(* Logix 5000 project; controller Receptivo vendor 1 type 14 code 106 rev 30.11; software revision 30.00; part 2 of 10 *)

        [54].Fecha.Minuto := 54, [54].Fecha.Segundo := 41, [54].Fecha.Milisegundos := 45401, [54].Lote := 147, [54].Operador := 5, [54].Descripcion := 'Alegria Caja 6 x 3000 cm3  - Costa', [54].EAN14 := '17702161043987', [54].QAD := '600300', [54].Peso_Real := 516.0, [54].Peso_Teorico := 519.0, [54].No_Cajas := 30, [54].Consec := 188, [54].Envase := 3000, [54].Envases_x_Caja := 6, [54].Densidad_Medida := 0.9152, [54].Linea := 3, [55].Fecha.year := 2021, [55].Fecha.Mes := 5, [55].Fecha.Dia := 27, [55].Fecha.Hora := 19, [55].Fecha.Minuto := 57, [55].Fecha.Segundo := 29, [55].Fecha.Milisegundos := 629132, [55].Lote := 147, [55].Operador := 5, [55].Descripcion := 'Alegria Caja 6 x 3000 cm3  - Costa', [55].EAN14 := '17702161043987', [55].QAD := '600300', [55].Peso_Real := 516.0, [55].Peso_Teorico := 519.0, [55].No_Cajas := 30, [55].Consec := 189, [55].Envase := 3000, [55].Envases_x_Caja := 6, [55].Densidad_Medida := 0.9152, [55].Linea := 3, [56].Fecha.year := 2021, [56].Fecha.Mes := 5, [56].Fecha.Dia := 27, [56].Fecha.Hora := 20, [56].Fecha.Segundo := 42, [56].Fecha.Milisegundos := 662176, [56].Lote := 147, [56].Operador := 5, [56].Descripcion := 'Alegria Caja 6 x 3000 cm3  - Costa', [56].EAN14 := '17702161043987', [56].QAD := '600300', [56].Peso_Real := 518.0, [56].Peso_Teorico := 519.0, [56].No_Cajas := 30, [56].Consec := 190, [56].Envase := 3000, [56].Envases_x_Caja := 6, [56].Densidad_Medida := 0.9152, [56].Linea := 3, [57].Fecha.year := 2021, [57].Fecha.Mes := 5, [57].Fecha.Dia := 27, [57].Fecha.Hora := 20, [57].Fecha.Minuto := 5,
        [57].Fecha.Segundo := 2, [57].Fecha.Milisegundos := 990759, [57].Lote := 147, [57].Operador := 5, [57].Descripcion := 'Alegria Caja 6 x 3000 cm3  - Costa', [57].EAN14 := '17702161043987', [57].QAD := '600300', [57].Peso_Real := 518.0, [57].Peso_Teorico := 519.0, [57].No_Cajas := 30, [57].Consec := 191, [57].Envase := 3000, [57].Envases_x_Caja := 6, [57].Densidad_Medida := 0.9152, [57].Linea := 3, [58].Fecha.year := 2021, [58].Fecha.Mes := 5, [58].Fecha.Dia := 27, [58].Fecha.Hora := 20, [58].Fecha.Minuto := 7, [58].Fecha.Segundo := 7, [58].Fecha.Milisegundos := 884753, [58].Lote := 147, [58].Operador := 5, [58].Descripcion := 'Alegria Caja 6 x 3000 cm3  - Costa', [58].EAN14 := '17702161043987', [58].QAD := '600300', [58].Peso_Real := 52.0, [58].Peso_Teorico := 52.0, [58].No_Cajas := 3, [58].Consec := 192, [58].Envase := 3000, [58].Envases_x_Caja := 6, [58].Densidad_Medida := 0.9152, [58].Linea := 3);
   Cola_Estacion_4 : UDT_COLA[100] := ([0].Fecha.year := 2021, [0].Fecha.Mes := 5, [0].Fecha.Dia := 28, [0].Fecha.Hora := 8, [0].Fecha.Minuto := 20, [0].Fecha.Segundo := 37, [0].Fecha.Milisegundos := 69124, [0].Lote := 148, [0].Operador := 6, [0].Descripcion := 'Aceite Vegetal Torino  Exp.', [0].EAN14 := '17702161820113', [0].QAD := '607020', [0].Peso_Real := 790.0, [0].Peso_Teorico := 786.0, [0].No_Cajas := 48, [0].Consec := 1, [0].Envase := 17250, [0].Envases_x_Caja := 1, [0].Densidad_Medida := 0.9148, [0].Linea := 5, [1].Fecha.year := 2021, [1].Fecha.Mes := 5, [1].Fecha.Dia := 28, [1].Fecha.Hora := 8, [1].Fecha.Minuto := 26, [1].Fecha.Segundo := 16, [1].Fecha.Milisegundos := 465551, [1].Lote := 148, [1].Operador := 6, [1].Descripcion := 'Aceite Vegetal Torino  Exp.', [1].EAN14 := '17702161820113', [1].QAD := '607020', [1].Peso_Real := 787.0, [1].Peso_Teorico := 786.0, [1].No_Cajas := 48, [1].Consec := 2, [1].Envase := 17250, [1].Envases_x_Caja := 1, [1].Densidad_Medida := 0.9148, [1].Linea := 5, [2].Fecha.year := 2021, [2].Fecha.Mes := 5, [2].Fecha.Dia := 28, [2].Fecha.Hora := 8, [2].Fecha.Minuto := 31, [2].Fecha.Segundo := 21, [2].Fecha.Milisegundos := 483752, [2].Lote := 148, [2].Operador := 6, [2].Descripcion := 'Aceite Vegetal Torino  Exp.', [2].EAN14 := '17702161820113', [2].QAD := '607020', [2].Peso_Real := 789.0, [2].Peso_Teorico := 786.0, [2].No_Cajas := 48, [2].Consec := 3, [2].Envase := 17250, [2].Envases_x_Caja := 1, [2].Densidad_Medida := 0.9148, [2].Linea := 5,
        [3].Fecha.year := 2021, [3].Fecha.Mes := 5, [3].Fecha.Dia := 28, [3].Fecha.Hora := 8, [3].Fecha.Minuto := 36, [3].Fecha.Segundo := 10, [3].Fecha.Milisegundos := 577902, [3].Lote := 148, [3].Operador := 6, [3].Descripcion := 'Aceite Vegetal Torino  Exp.', [3].EAN14 := '17702161820113', [3].QAD := '607020', [3].Peso_Real := 786.0, [3].Peso_Teorico := 786.0, [3].No_Cajas := 48, [3].Consec := 4, [3].Envase := 17250, [3].Envases_x_Caja := 1, [3].Densidad_Medida := 0.9148, [3].Linea := 5, [4].Fecha.year := 2021, [4].Fecha.Mes := 5, [4].Fecha.Dia := 28, [4].Fecha.Hora := 8, [4].Fecha.Minuto := 40, [4].Fecha.Segundo := 51, [4].Fecha.Milisegundos := 336954, [4].Lote := 148, [4].Operador := 6, [4].Descripcion := 'Aceite Vegetal Torino  Exp.', [4].EAN14 := '17702161820113', [4].QAD := '607020', [4].Peso_Real := 790.0, [4].Peso_Teorico := 786.0, [4].No_Cajas := 48, [4].Consec := 5, [4].Envase := 17250, [4].Envases_x_Caja := 1, [4].Densidad_Medida := 0.9148, [4].Linea := 5, [5].Fecha.year := 2021, [5].Fecha.Mes := 5, [5].Fecha.Dia := 28, [5].Fecha.Hora := 8, [5].Fecha.Minuto := 47, [5].Fecha.Segundo := 15, [5].Fecha.Milisegundos := 315402, [5].Lote := 148, [5].Operador := 6, [5].Descripcion := 'Aceite Vegetal Torino  Exp.', [5].EAN14 := '17702161820113', [5].QAD := '607020', [5].Peso_Real := 789.0, [5].Peso_Teorico := 786.0, [5].No_Cajas := 48, [5].Consec := 6, [5].Envase := 17250, [5].Envases_x_Caja := 1, [5].Densidad_Medida := 0.9148, [5].Linea := 5,
        [6].Fecha.year := 2021, [6].Fecha.Mes := 5, [6].Fecha.Dia := 28, [6].Fecha.Hora := 8, [6].Fecha.Minuto := 52, [6].Fecha.Segundo := 9, [6].Fecha.Milisegundos := 719173, [6].Lote := 148, [6].Operador := 6, [6].Descripcion := 'Aceite Vegetal Torino  Exp.', [6].EAN14 := '17702161820113', [6].QAD := '607020', [6].Peso_Real := 787.0, [6].Peso_Teorico := 786.0, [6].No_Cajas := 48, [6].Consec := 7, [6].Envase := 17250, [6].Envases_x_Caja := 1, [6].Densidad_Medida := 0.9148, [6].Linea := 5, [7].Fecha.year := 2021, [7].Fecha.Mes := 5, [7].Fecha.Dia := 28, [7].Fecha.Hora := 8, [7].Fecha.Minuto := 55, [7].Fecha.Segundo := 40, [7].Fecha.Milisegundos := 508565, [7].Lote := 148, [7].Operador := 6, [7].Descripcion := 'Aceite Vegetal Torino  Exp.', [7].EAN14 := '17702161820113', [7].QAD := '607020', [7].Peso_Real := 791.0, [7].Peso_Teorico := 786.0, [7].No_Cajas := 48, [7].Consec := 8, [7].Envase := 17250, [7].Envases_x_Caja := 1, [7].Densidad_Medida := 0.9148, [7].Linea := 5, [8].Fecha.year := 2021, [8].Fecha.Mes := 5, [8].Fecha.Dia := 28, [8].Fecha.Hora := 9, [8].Fecha.Segundo := 2, [8].Fecha.Milisegundos := 670788, [8].Lote := 148, [8].Operador := 6, [8].Descripcion := 'Aceite Vegetal Torino  Exp.', [8].EAN14 := '17702161820113', [8].QAD := '607020', [8].Peso_Real := 789.0, [8].Peso_Teorico := 786.0, [8].No_Cajas := 48, [8].Consec := 9, [8].Envase := 17250, [8].Envases_x_Caja := 1, [8].Densidad_Medida := 0.9148, [8].Linea := 5, [9].Fecha.year := 2021,
        [9].Fecha.Mes := 5, [9].Fecha.Dia := 28, [9].Fecha.Hora := 9, [9].Fecha.Minuto := 4, [9].Fecha.Segundo := 22, [9].Fecha.Milisegundos := 670540, [9].Lote := 148, [9].Operador := 6, [9].Descripcion := 'Aceite Vegetal Torino  Exp.', [9].EAN14 := '17702161820113', [9].QAD := '607020', [9].Peso_Real := 788.0, [9].Peso_Teorico := 786.0, [9].No_Cajas := 48, [9].Consec := 10, [9].Envase := 17250, [9].Envases_x_Caja := 1, [9].Densidad_Medida := 0.9148, [9].Linea := 5, [10].Fecha.year := 2021, [10].Fecha.Mes := 5, [10].Fecha.Dia := 28, [10].Fecha.Hora := 9, [10].Fecha.Minuto := 12, [10].Fecha.Segundo := 17, [10].Fecha.Milisegundos := 553199, [10].Lote := 148, [10].Operador := 6, [10].Descripcion := 'Aceite Vegetal Torino  Exp.', [10].EAN14 := '17702161820113', [10].QAD := '607020', [10].Peso_Real := 787.0, [10].Peso_Teorico := 786.0, [10].No_Cajas := 48, [10].Consec := 11, [10].Envase := 17250, [10].Envases_x_Caja := 1, [10].Densidad_Medida := 0.9148, [10].Linea := 5, [11].Fecha.year := 2021, [11].Fecha.Mes := 5, [11].Fecha.Dia := 28, [11].Fecha.Hora := 9, [11].Fecha.Minuto := 17, [11].Fecha.Segundo := 9, [11].Fecha.Milisegundos := 930477, [11].Lote := 148, [11].Operador := 6, [11].Descripcion := 'Aceite Vegetal Torino  Exp.', [11].EAN14 := '17702161820113', [11].QAD := '607020', [11].Peso_Real := 787.0, [11].Peso_Teorico := 786.0, [11].No_Cajas := 48, [11].Consec := 12, [11].Envase := 17250, [11].Envases_x_Caja := 1, [11].Densidad_Medida := 0.9148, [11].Linea := 5, [12].Fecha.year := 2021,
        [12].Fecha.Mes := 5, [12].Fecha.Dia := 28, [12].Fecha.Hora := 9, [12].Fecha.Minuto := 21, [12].Fecha.Segundo := 57, [12].Fecha.Milisegundos := 591967, [12].Lote := 148, [12].Operador := 6, [12].Descripcion := 'Aceite Vegetal Torino  Exp.', [12].EAN14 := '17702161820113', [12].QAD := '607020', [12].Peso_Real := 787.0, [12].Peso_Teorico := 786.0, [12].No_Cajas := 48, [12].Consec := 13, [12].Envase := 17250, [12].Envases_x_Caja := 1, [12].Densidad_Medida := 0.9148, [12].Linea := 5, [13].Fecha.year := 2021, [13].Fecha.Mes := 5, [13].Fecha.Dia := 28, [13].Fecha.Hora := 9, [13].Fecha.Minuto := 26, [13].Fecha.Segundo := 49, [13].Fecha.Milisegundos := 73835, [13].Lote := 148, [13].Operador := 6, [13].Descripcion := 'Aceite Vegetal Torino  Exp.', [13].EAN14 := '17702161820113', [13].QAD := '607020', [13].Peso_Real := 786.0, [13].Peso_Teorico := 786.0, [13].No_Cajas := 48, [13].Consec := 14, [13].Envase := 17250, [13].Envases_x_Caja := 1, [13].Densidad_Medida := 0.9148, [13].Linea := 5, [14].Fecha.year := 2021, [14].Fecha.Mes := 5, [14].Fecha.Dia := 28, [14].Fecha.Hora := 9, [14].Fecha.Minuto := 32, [14].Fecha.Segundo := 14, [14].Fecha.Milisegundos := 130378, [14].Lote := 148, [14].Operador := 6, [14].Descripcion := 'Aceite Vegetal Torino  Exp.', [14].EAN14 := '17702161820113', [14].QAD := '607020', [14].Peso_Real := 786.0, [14].Peso_Teorico := 786.0, [14].No_Cajas := 48, [14].Consec := 15, [14].Envase := 17250, [14].Envases_x_Caja := 1, [14].Densidad_Medida := 0.9148, [14].Linea := 5, [15].Fecha.year := 2021,
        [15].Fecha.Mes := 5, [15].Fecha.Dia := 28, [15].Fecha.Hora := 9, [15].Fecha.Minuto := 38, [15].Fecha.Segundo := 57, [15].Fecha.Milisegundos := 869726, [15].Lote := 148, [15].Operador := 6, [15].Descripcion := 'Aceite Vegetal Torino  Exp.', [15].EAN14 := '17702161820113', [15].QAD := '607020', [15].Peso_Real := 789.0, [15].Peso_Teorico := 786.0, [15].No_Cajas := 48, [15].Consec := 16, [15].Envase := 17250, [15].Envases_x_Caja := 1, [15].Densidad_Medida := 0.9148, [15].Linea := 5, [16].Fecha.year := 2021, [16].Fecha.Mes := 5, [16].Fecha.Dia := 28, [16].Fecha.Hora := 9, [16].Fecha.Minuto := 43, [16].Fecha.Segundo := 25, [16].Fecha.Milisegundos := 20130, [16].Lote := 148, [16].Operador := 6, [16].Descripcion := 'Aceite Vegetal Torino  Exp.', [16].EAN14 := '17702161820113', [16].QAD := '607020', [16].Peso_Real := 790.0, [16].Peso_Teorico := 786.0, [16].No_Cajas := 48, [16].Consec := 17, [16].Envase := 17250, [16].Envases_x_Caja := 1, [16].Densidad_Medida := 0.9148, [16].Linea := 5, [17].Fecha.year := 2021, [17].Fecha.Mes := 5, [17].Fecha.Dia := 28, [17].Fecha.Hora := 9, [17].Fecha.Minuto := 47, [17].Fecha.Segundo := 58, [17].Fecha.Milisegundos := 358560, [17].Lote := 148, [17].Operador := 6, [17].Descripcion := 'Aceite Vegetal Torino  Exp.', [17].EAN14 := '17702161820113', [17].QAD := '607020', [17].Peso_Real := 789.0, [17].Peso_Teorico := 786.0, [17].No_Cajas := 48, [17].Consec := 18, [17].Envase := 17250, [17].Envases_x_Caja := 1, [17].Densidad_Medida := 0.9148, [17].Linea := 5, [18].Fecha.year := 2021,
        [18].Fecha.Mes := 5, [18].Fecha.Dia := 28, [18].Fecha.Hora := 9, [18].Fecha.Minuto := 51, [18].Fecha.Segundo := 17, [18].Fecha.Milisegundos := 179162, [18].Lote := 148, [18].Operador := 6, [18].Descripcion := 'Aceite Vegetal Torino  Exp.', [18].EAN14 := '17702161820113', [18].QAD := '607020', [18].Peso_Real := 788.0, [18].Peso_Teorico := 786.0, [18].No_Cajas := 48, [18].Consec := 19, [18].Envase := 17250, [18].Envases_x_Caja := 1, [18].Densidad_Medida := 0.9148, [18].Linea := 5, [19].Fecha.year := 2021, [19].Fecha.Mes := 5, [19].Fecha.Dia := 28, [19].Fecha.Hora := 9, [19].Fecha.Minuto := 54, [19].Fecha.Segundo := 47, [19].Fecha.Milisegundos := 964537, [19].Lote := 148, [19].Operador := 6, [19].Descripcion := 'Aceite Vegetal Torino  Exp.', [19].EAN14 := '17702161820113', [19].QAD := '607020', [19].Peso_Real := 788.0, [19].Peso_Teorico := 786.0, [19].No_Cajas := 48, [19].Consec := 20, [19].Envase := 17250, [19].Envases_x_Caja := 1, [19].Densidad_Medida := 0.9148, [19].Linea := 5, [20].Fecha.year := 2021, [20].Fecha.Mes := 5, [20].Fecha.Dia := 28, [20].Fecha.Hora := 10, [20].Fecha.Minuto := 3, [20].Fecha.Segundo := 29, [20].Fecha.Milisegundos := 988763, [20].Lote := 148, [20].Operador := 6, [20].Descripcion := 'Aceite Vegetal Torino  Exp.', [20].EAN14 := '17702161820113', [20].QAD := '607020', [20].Peso_Real := 787.0, [20].Peso_Teorico := 786.0, [20].No_Cajas := 48, [20].Consec := 21, [20].Envase := 17250, [20].Envases_x_Caja := 1, [20].Densidad_Medida := 0.9148, [20].Linea := 5, [21].Fecha.year := 2021,
        [21].Fecha.Mes := 5, [21].Fecha.Dia := 28, [21].Fecha.Hora := 10, [21].Fecha.Minuto := 9, [21].Fecha.Segundo := 7, [21].Fecha.Milisegundos := 475825, [21].Lote := 148, [21].Operador := 6, [21].Descripcion := 'Aceite Vegetal Torino  Exp.', [21].EAN14 := '17702161820113', [21].QAD := '607020', [21].Peso_Real := 788.0, [21].Peso_Teorico := 786.0, [21].No_Cajas := 48, [21].Consec := 22, [21].Envase := 17250, [21].Envases_x_Caja := 1, [21].Densidad_Medida := 0.9148, [21].Linea := 5, [22].Fecha.year := 2021, [22].Fecha.Mes := 5, [22].Fecha.Dia := 28, [22].Fecha.Hora := 10, [22].Fecha.Minuto := 13, [22].Fecha.Segundo := 59, [22].Fecha.Milisegundos := 393945, [22].Lote := 148, [22].Operador := 6, [22].Descripcion := 'Aceite Vegetal Torino  Exp.', [22].EAN14 := '17702161820113', [22].QAD := '607020', [22].Peso_Real := 788.0, [22].Peso_Teorico := 786.0, [22].No_Cajas := 48, [22].Consec := 23, [22].Envase := 17250, [22].Envases_x_Caja := 1, [22].Densidad_Medida := 0.9148, [22].Linea := 5, [23].Fecha.year := 2021, [23].Fecha.Mes := 5, [23].Fecha.Dia := 28, [23].Fecha.Hora := 10, [23].Fecha.Minuto := 18, [23].Fecha.Segundo := 56, [23].Fecha.Milisegundos := 553433, [23].Lote := 148, [23].Operador := 6, [23].Descripcion := 'Aceite Vegetal Torino  Exp.', [23].EAN14 := '17702161820113', [23].QAD := '607020', [23].Peso_Real := 787.0, [23].Peso_Teorico := 786.0, [23].No_Cajas := 48, [23].Consec := 24, [23].Envase := 17250, [23].Envases_x_Caja := 1, [23].Densidad_Medida := 0.9148, [23].Linea := 5, [24].Fecha.year := 2021,
        [24].Fecha.Mes := 5, [24].Fecha.Dia := 28, [24].Fecha.Hora := 10, [24].Fecha.Minuto := 24, [24].Fecha.Segundo := 26, [24].Fecha.Milisegundos := 21235, [24].Lote := 148, [24].Operador := 6, [24].Descripcion := 'Aceite Vegetal Torino  Exp.', [24].EAN14 := '17702161820113', [24].QAD := '607020', [24].Peso_Real := 787.0, [24].Peso_Teorico := 786.0, [24].No_Cajas := 48, [24].Consec := 25, [24].Envase := 17250, [24].Envases_x_Caja := 1, [24].Densidad_Medida := 0.9148, [24].Linea := 5, [25].Fecha.year := 2021, [25].Fecha.Mes := 5, [25].Fecha.Dia := 28, [25].Fecha.Hora := 10, [25].Fecha.Minuto := 30, [25].Fecha.Segundo := 54, [25].Fecha.Milisegundos := 336113, [25].Lote := 148, [25].Operador := 6, [25].Descripcion := 'Aceite Vegetal Torino  Exp.', [25].EAN14 := '17702161820113', [25].QAD := '607020', [25].Peso_Real := 790.0, [25].Peso_Teorico := 786.0, [25].No_Cajas := 48, [25].Consec := 26, [25].Envase := 17250, [25].Envases_x_Caja := 1, [25].Densidad_Medida := 0.9148, [25].Linea := 5, [26].Fecha.year := 2021, [26].Fecha.Mes := 5, [26].Fecha.Dia := 28, [26].Fecha.Hora := 10, [26].Fecha.Minuto := 35, [26].Fecha.Segundo := 32, [26].Fecha.Milisegundos := 418041, [26].Lote := 148, [26].Operador := 6, [26].Descripcion := 'Aceite Vegetal Torino  Exp.', [26].EAN14 := '17702161820113', [26].QAD := '607020', [26].Peso_Real := 789.0, [26].Peso_Teorico := 786.0, [26].No_Cajas := 48, [26].Consec := 27, [26].Envase := 17250, [26].Envases_x_Caja := 1, [26].Densidad_Medida := 0.9148, [26].Linea := 5, [27].Fecha.year := 2021,
        [27].Fecha.Mes := 5, [27].Fecha.Dia := 28, [27].Fecha.Hora := 10, [27].Fecha.Minuto := 40, [27].Fecha.Segundo := 38, [27].Fecha.Milisegundos := 622882, [27].Lote := 148, [27].Operador := 6, [27].Descripcion := 'Aceite Vegetal Torino  Exp.', [27].EAN14 := '17702161820113', [27].QAD := '607020', [27].Peso_Real := 794.0, [27].Peso_Teorico := 786.0, [27].No_Cajas := 48, [27].Consec := 28, [27].Envase := 17250, [27].Envases_x_Caja := 1, [27].Densidad_Medida := 0.9148, [27].Linea := 5, [28].Fecha.year := 2021, [28].Fecha.Mes := 5, [28].Fecha.Dia := 28, [28].Fecha.Hora := 10, [28].Fecha.Minuto := 45, [28].Fecha.Segundo := 3, [28].Fecha.Milisegundos := 533526, [28].Lote := 148, [28].Operador := 6, [28].Descripcion := 'Aceite Vegetal Torino  Exp.', [28].EAN14 := '17702161820113', [28].QAD := '607020', [28].Peso_Real := 791.0, [28].Peso_Teorico := 786.0, [28].No_Cajas := 48, [28].Consec := 29, [28].Envase := 17250, [28].Envases_x_Caja := 1, [28].Densidad_Medida := 0.9148, [28].Linea := 5, [29].Fecha.year := 2021, [29].Fecha.Mes := 5, [29].Fecha.Dia := 28, [29].Fecha.Hora := 10, [29].Fecha.Minuto := 49, [29].Fecha.Segundo := 29, [29].Fecha.Milisegundos := 771525, [29].Lote := 148, [29].Operador := 6, [29].Descripcion := 'Aceite Vegetal Torino  Exp.', [29].EAN14 := '17702161820113', [29].QAD := '607020', [29].Peso_Real := 789.0, [29].Peso_Teorico := 786.0, [29].No_Cajas := 48, [29].Consec := 30, [29].Envase := 17250, [29].Envases_x_Caja := 1, [29].Densidad_Medida := 0.9148, [29].Linea := 5, [30].Fecha.year := 2021,
        [30].Fecha.Mes := 5, [30].Fecha.Dia := 28, [30].Fecha.Hora := 11, [30].Fecha.Minuto := 38, [30].Fecha.Segundo := 27, [30].Fecha.Milisegundos := 412017, [30].Lote := 148, [30].Operador := 6, [30].Descripcion := 'Aceite Vegetal Torino  Exp.', [30].EAN14 := '17702161820113', [30].QAD := '607020', [30].Peso_Real := 787.0, [30].Peso_Teorico := 786.0, [30].No_Cajas := 48, [30].Consec := 37, [30].Envase := 17250, [30].Envases_x_Caja := 1, [30].Densidad_Medida := 0.9148, [30].Linea := 5, [31].Fecha.year := 2021, [31].Fecha.Mes := 5, [31].Fecha.Dia := 28, [31].Fecha.Hora := 11, [31].Fecha.Minuto := 43, [31].Fecha.Segundo := 1, [31].Fecha.Milisegundos := 735545, [31].Lote := 148, [31].Operador := 6, [31].Descripcion := 'Aceite Vegetal Torino  Exp.', [31].EAN14 := '17702161820113', [31].QAD := '607020', [31].Peso_Real := 787.0, [31].Peso_Teorico := 786.0, [31].No_Cajas := 48, [31].Consec := 39, [31].Envase := 17250, [31].Envases_x_Caja := 1, [31].Densidad_Medida := 0.9148, [31].Linea := 5, [32].Fecha.year := 2021, [32].Fecha.Mes := 5, [32].Fecha.Dia := 28, [32].Fecha.Hora := 11, [32].Fecha.Minuto := 47, [32].Fecha.Segundo := 48, [32].Fecha.Milisegundos := 728105, [32].Lote := 148, [32].Operador := 6, [32].Descripcion := 'Aceite Vegetal Torino  Exp.', [32].EAN14 := '17702161820113', [32].QAD := '607020', [32].Peso_Real := 787.0, [32].Peso_Teorico := 786.0, [32].No_Cajas := 48, [32].Consec := 42, [32].Envase := 17250, [32].Envases_x_Caja := 1, [32].Densidad_Medida := 0.9148, [32].Linea := 5, [33].Fecha.year := 2021,
        [33].Fecha.Mes := 5, [33].Fecha.Dia := 28, [33].Fecha.Hora := 11, [33].Fecha.Minuto := 54, [33].Fecha.Segundo := 28, [33].Fecha.Milisegundos := 332631, [33].Lote := 148, [33].Operador := 6, [33].Descripcion := 'Aceite Vegetal Torino  Exp.', [33].EAN14 := '17702161820113', [33].QAD := '607020', [33].Peso_Real := 788.0, [33].Peso_Teorico := 786.0, [33].No_Cajas := 48, [33].Consec := 46, [33].Envase := 17250, [33].Envases_x_Caja := 1, [33].Densidad_Medida := 0.9148, [33].Linea := 5, [34].Fecha.year := 2021, [34].Fecha.Mes := 5, [34].Fecha.Dia := 28, [34].Fecha.Hora := 12, [34].Fecha.Minuto := 37, [34].Fecha.Segundo := 29, [34].Fecha.Milisegundos := 409886, [34].Lote := 148, [34].Operador := 6, [34].Descripcion := 'Aceite Vegetal Torino  Exp.', [34].EAN14 := '17702161820113', [34].QAD := '607020', [34].Peso_Real := 789.0, [34].Peso_Teorico := 786.0, [34].No_Cajas := 48, [34].Consec := 61, [34].Envase := 17250, [34].Envases_x_Caja := 1, [34].Densidad_Medida := 0.9148, [34].Linea := 5, [35].Fecha.year := 2021, [35].Fecha.Mes := 5, [35].Fecha.Dia := 28, [35].Fecha.Hora := 12, [35].Fecha.Minuto := 48, [35].Fecha.Segundo := 16, [35].Fecha.Milisegundos := 558137, [35].Lote := 148, [35].Operador := 6, [35].Descripcion := 'Aceite Vegetal Torino  Exp.', [35].EAN14 := '17702161820113', [35].QAD := '607020', [35].Peso_Real := 788.0, [35].Peso_Teorico := 786.0, [35].No_Cajas := 48, [35].Consec := 64, [35].Envase := 17250, [35].Envases_x_Caja := 1, [35].Densidad_Medida := 0.9148, [35].Linea := 5, [36].Fecha.year := 2021,
        [36].Fecha.Mes := 5, [36].Fecha.Dia := 28, [36].Fecha.Hora := 12, [36].Fecha.Minuto := 53, [36].Fecha.Segundo := 29, [36].Fecha.Milisegundos := 332540, [36].Lote := 148, [36].Operador := 6, [36].Descripcion := 'Aceite Vegetal Torino  Exp.', [36].EAN14 := '17702161820113', [36].QAD := '607020', [36].Peso_Real := 790.0, [36].Peso_Teorico := 786.0, [36].No_Cajas := 48, [36].Consec := 66, [36].Envase := 17250, [36].Envases_x_Caja := 1, [36].Densidad_Medida := 0.9148, [36].Linea := 5, [37].Fecha.year := 2021, [37].Fecha.Mes := 5, [37].Fecha.Dia := 28, [37].Fecha.Hora := 12, [37].Fecha.Minuto := 59, [37].Fecha.Segundo := 39, [37].Fecha.Milisegundos := 67313, [37].Lote := 148, [37].Operador := 6, [37].Descripcion := 'Aceite Vegetal Torino  Exp.', [37].EAN14 := '17702161820113', [37].QAD := '607020', [37].Peso_Real := 784.0, [37].Peso_Teorico := 786.0, [37].No_Cajas := 48, [37].Consec := 68, [37].Envase := 17250, [37].Envases_x_Caja := 1, [37].Densidad_Medida := 0.9148, [37].Linea := 5, [38].Fecha.year := 2021, [38].Fecha.Mes := 5, [38].Fecha.Dia := 28, [38].Fecha.Hora := 13, [38].Fecha.Minuto := 4, [38].Fecha.Segundo := 44, [38].Fecha.Milisegundos := 914365, [38].Lote := 148, [38].Operador := 6, [38].Descripcion := 'Aceite Vegetal Torino  Exp.', [38].EAN14 := '17702161820113', [38].QAD := '607020', [38].Peso_Real := 788.0, [38].Peso_Teorico := 786.0, [38].No_Cajas := 48, [38].Consec := 70, [38].Envase := 17250, [38].Envases_x_Caja := 1, [38].Densidad_Medida := 0.9148, [38].Linea := 5, [39].Fecha.year := 2021,
        [39].Fecha.Mes := 5, [39].Fecha.Dia := 28, [39].Fecha.Hora := 13, [39].Fecha.Minuto := 9, [39].Fecha.Segundo := 50, [39].Fecha.Milisegundos := 10253, [39].Lote := 148, [39].Operador := 6, [39].Descripcion := 'Aceite Vegetal Torino  Exp.', [39].EAN14 := '17702161820113', [39].QAD := '607020', [39].Peso_Real := 788.0, [39].Peso_Teorico := 786.0, [39].No_Cajas := 48, [39].Consec := 73, [39].Envase := 17250, [39].Envases_x_Caja := 1, [39].Densidad_Medida := 0.9148, [39].Linea := 5, [40].Fecha.year := 2021, [40].Fecha.Mes := 5, [40].Fecha.Dia := 28, [40].Fecha.Hora := 13, [40].Fecha.Minuto := 18, [40].Fecha.Segundo := 54, [40].Fecha.Milisegundos := 825126, [40].Lote := 148, [40].Operador := 6, [40].Descripcion := 'Aceite Vegetal Torino  Exp.', [40].EAN14 := '17702161820113', [40].QAD := '607020', [40].Peso_Real := 790.0, [40].Peso_Teorico := 786.0, [40].No_Cajas := 48, [40].Consec := 78, [40].Envase := 17250, [40].Envases_x_Caja := 1, [40].Densidad_Medida := 0.9148, [40].Linea := 5, [41].Fecha.year := 2021, [41].Fecha.Mes := 5, [41].Fecha.Dia := 28, [41].Fecha.Hora := 13, [41].Fecha.Minuto := 23, [41].Fecha.Segundo := 24, [41].Fecha.Milisegundos := 204408, [41].Lote := 148, [41].Operador := 6, [41].Descripcion := 'Aceite Vegetal Torino  Exp.', [41].EAN14 := '17702161820113', [41].QAD := '607020', [41].Peso_Real := 790.0, [41].Peso_Teorico := 786.0, [41].No_Cajas := 48, [41].Consec := 81, [41].Envase := 17250, [41].Envases_x_Caja := 1, [41].Densidad_Medida := 0.9148, [41].Linea := 5, [42].Fecha.year := 2021,
        [42].Fecha.Mes := 5, [42].Fecha.Dia := 28, [42].Fecha.Hora := 13, [42].Fecha.Minuto := 28, [42].Fecha.Segundo := 7, [42].Fecha.Milisegundos := 125838, [42].Lote := 148, [42].Operador := 6, [42].Descripcion := 'Aceite Vegetal Torino  Exp.', [42].EAN14 := '17702161820113', [42].QAD := '607020', [42].Peso_Real := 787.0, [42].Peso_Teorico := 786.0, [42].No_Cajas := 48, [42].Consec := 84, [42].Envase := 17250, [42].Envases_x_Caja := 1, [42].Densidad_Medida := 0.9148, [42].Linea := 5, [43].Fecha.year := 2021, [43].Fecha.Mes := 5, [43].Fecha.Dia := 28, [43].Fecha.Hora := 13, [43].Fecha.Minuto := 34, [43].Fecha.Segundo := 9, [43].Fecha.Milisegundos := 399329, [43].Lote := 148, [43].Operador := 6, [43].Descripcion := 'Aceite Vegetal Torino  Exp.', [43].EAN14 := '17702161820113', [43].QAD := '607020', [43].Peso_Real := 788.0, [43].Peso_Teorico := 786.0, [43].No_Cajas := 48, [43].Consec := 87, [43].Envase := 17250, [43].Envases_x_Caja := 1, [43].Densidad_Medida := 0.9148, [43].Linea := 5, [44].Fecha.year := 2021, [44].Fecha.Mes := 5, [44].Fecha.Dia := 28, [44].Fecha.Hora := 13, [44].Fecha.Minuto := 42, [44].Fecha.Segundo := 2, [44].Fecha.Milisegundos := 643055, [44].Lote := 148, [44].Operador := 6, [44].Descripcion := 'Aceite Vegetal Torino  Exp.', [44].EAN14 := '17702161820113', [44].QAD := '607020', [44].Peso_Real := 791.0, [44].Peso_Teorico := 786.0, [44].No_Cajas := 48, [44].Consec := 88, [44].Envase := 17250, [44].Envases_x_Caja := 1, [44].Densidad_Medida := 0.9148, [44].Linea := 5, [45].Fecha.year := 2021,
        [45].Fecha.Mes := 5, [45].Fecha.Dia := 28, [45].Fecha.Hora := 13, [45].Fecha.Minuto := 54, [45].Fecha.Segundo := 53, [45].Fecha.Milisegundos := 530969, [45].Lote := 148, [45].Operador := 6, [45].Descripcion := 'Aceite Vegetal Torino  Exp.', [45].EAN14 := '17702161820113', [45].QAD := '607020', [45].Peso_Real := 792.0, [45].Peso_Teorico := 786.0, [45].No_Cajas := 48, [45].Consec := 90, [45].Envase := 17250, [45].Envases_x_Caja := 1, [45].Densidad_Medida := 0.9148, [45].Linea := 5, [46].Fecha.year := 2021, [46].Fecha.Mes := 5, [46].Fecha.Dia := 28, [46].Fecha.Hora := 14, [46].Fecha.Minuto := 1, [46].Fecha.Segundo := 32, [46].Fecha.Milisegundos := 314203, [46].Lote := 148, [46].Operador := 6, [46].Descripcion := 'Aceite Vegetal Torino  Exp.', [46].EAN14 := '17702161820113', [46].QAD := '607020', [46].Peso_Real := 786.0, [46].Peso_Teorico := 786.0, [46].No_Cajas := 48, [46].Consec := 94, [46].Envase := 17250, [46].Envases_x_Caja := 1, [46].Densidad_Medida := 0.9148, [46].Linea := 5, [47].Fecha.year := 2021, [47].Fecha.Mes := 5, [47].Fecha.Dia := 28, [47].Fecha.Hora := 14, [47].Fecha.Minuto := 13, [47].Fecha.Segundo := 9, [47].Fecha.Milisegundos := 540121, [47].Lote := 148, [47].Operador := 6, [47].Descripcion := 'Aceite Vegetal Torino  Exp.', [47].EAN14 := '17702161820113', [47].QAD := '607020', [47].Peso_Real := 787.0, [47].Peso_Teorico := 786.0, [47].No_Cajas := 48, [47].Consec := 98, [47].Envase := 17250, [47].Envases_x_Caja := 1, [47].Densidad_Medida := 0.9148, [47].Linea := 5, [48].Fecha.year := 2021,
        [48].Fecha.Mes := 5, [48].Fecha.Dia := 28, [48].Fecha.Hora := 14, [48].Fecha.Minuto := 20, [48].Fecha.Segundo := 32, [48].Fecha.Milisegundos := 366895, [48].Lote := 148, [48].Operador := 6, [48].Descripcion := 'Aceite Vegetal Torino  Exp.', [48].EAN14 := '17702161820113', [48].QAD := '607020', [48].Peso_Real := 788.0, [48].Peso_Teorico := 786.0, [48].No_Cajas := 48, [48].Consec := 102, [48].Envase := 17250, [48].Envases_x_Caja := 1, [48].Densidad_Medida := 0.9148, [48].Linea := 5, [49].Fecha.year := 2021, [49].Fecha.Mes := 5, [49].Fecha.Dia := 28, [49].Fecha.Hora := 14, [49].Fecha.Minuto := 25, [49].Fecha.Segundo := 56, [49].Fecha.Milisegundos := 412691, [49].Lote := 148, [49].Operador := 6, [49].Descripcion := 'Aceite Vegetal Torino  Exp.', [49].EAN14 := '17702161820113', [49].QAD := '607020', [49].Peso_Real := 789.0, [49].Peso_Teorico := 786.0, [49].No_Cajas := 48, [49].Consec := 103, [49].Envase := 17250, [49].Envases_x_Caja := 1, [49].Densidad_Medida := 0.9148, [49].Linea := 5, [50].Fecha.year := 2021, [50].Fecha.Mes := 5, [50].Fecha.Dia := 28, [50].Fecha.Hora := 14, [50].Fecha.Minuto := 34, [50].Fecha.Segundo := 53, [50].Fecha.Milisegundos := 121800, [50].Lote := 148, [50].Operador := 6, [50].Descripcion := 'Aceite Vegetal Torino  Exp.', [50].EAN14 := '17702161820113', [50].QAD := '607020', [50].Peso_Real := 786.0, [50].Peso_Teorico := 786.0, [50].No_Cajas := 48, [50].Consec := 106, [50].Envase := 17250, [50].Envases_x_Caja := 1, [50].Densidad_Medida := 0.9148, [50].Linea := 5, [51].Fecha.year := 2021,
        [51].Fecha.Mes := 5, [51].Fecha.Dia := 28, [51].Fecha.Hora := 14, [51].Fecha.Minuto := 41, [51].Fecha.Segundo := 59, [51].Fecha.Milisegundos := 904400, [51].Lote := 148, [51].Operador := 6, [51].Descripcion := 'Aceite Vegetal Torino  Exp.', [51].EAN14 := '17702161820113', [51].QAD := '607020', [51].Peso_Real := 789.0, [51].Peso_Teorico := 786.0, [51].No_Cajas := 48, [51].Consec := 108, [51].Envase := 17250, [51].Envases_x_Caja := 1, [51].Densidad_Medida := 0.9148, [51].Linea := 5, [52].Fecha.year := 2021, [52].Fecha.Mes := 5, [52].Fecha.Dia := 28, [52].Fecha.Hora := 14, [52].Fecha.Minuto := 49, [52].Fecha.Segundo := 25, [52].Fecha.Milisegundos := 216916, [52].Lote := 148, [52].Operador := 6, [52].Descripcion := 'Aceite Vegetal Torino  Exp.', [52].EAN14 := '17702161820113', [52].QAD := '607020', [52].Peso_Real := 787.0, [52].Peso_Teorico := 786.0, [52].No_Cajas := 48, [52].Consec := 110, [52].Envase := 17250, [52].Envases_x_Caja := 1, [52].Densidad_Medida := 0.9148, [52].Linea := 5);
   Cola_Estacion_4_A : UDT_COLA[100] := ([0].Fecha.year := 2021, [0].Fecha.Mes := 5, [0].Fecha.Dia := 27, [0].Fecha.Hora := 8, [0].Fecha.Minuto := 12, [0].Fecha.Segundo := 20, [0].Fecha.Milisegundos := 439054, [0].Lote := 147, [0].Operador := 6, [0].Descripcion := 'Aceite Vegetal Torino  Exp.', [0].EAN14 := '17702161820113', [0].QAD := '607020', [0].Peso_Real := 792.0, [0].Peso_Teorico := 786.0, [0].No_Cajas := 48, [0].Consec := 1, [0].Envase := 17250, [0].Envases_x_Caja := 1, [0].Densidad_Medida := 0.9148, [0].Linea := 5, [1].Fecha.year := 2021, [1].Fecha.Mes := 5, [1].Fecha.Dia := 27, [1].Fecha.Hora := 8, [1].Fecha.Minuto := 16, [1].Fecha.Segundo := 14, [1].Fecha.Milisegundos := 936761, [1].Lote := 147, [1].Operador := 6, [1].Descripcion := 'Aceite Vegetal Torino  Exp.', [1].EAN14 := '17702161820113', [1].QAD := '607020', [1].Peso_Real := 791.0, [1].Peso_Teorico := 786.0, [1].No_Cajas := 48, [1].Consec := 2, [1].Envase := 17250, [1].Envases_x_Caja := 1, [1].Densidad_Medida := 0.9148, [1].Linea := 5, [2].Fecha.year := 2021, [2].Fecha.Mes := 5, [2].Fecha.Dia := 27, [2].Fecha.Hora := 8, [2].Fecha.Minuto := 21, [2].Fecha.Segundo := 6, [2].Fecha.Milisegundos := 817817, [2].Lote := 147, [2].Operador := 6, [2].Descripcion := 'Aceite Vegetal Torino  Exp.', [2].EAN14 := '17702161820113', [2].QAD := '607020', [2].Peso_Real := 794.0, [2].Peso_Teorico := 786.0, [2].No_Cajas := 48, [2].Consec := 3, [2].Envase := 17250, [2].Envases_x_Caja := 1, [2].Densidad_Medida := 0.9148, [2].Linea := 5,
        [3].Fecha.year := 2021, [3].Fecha.Mes := 5, [3].Fecha.Dia := 27, [3].Fecha.Hora := 8, [3].Fecha.Minuto := 25, [3].Fecha.Segundo := 3, [3].Fecha.Milisegundos := 927147, [3].Lote := 147, [3].Operador := 6, [3].Descripcion := 'Aceite Vegetal Torino  Exp.', [3].EAN14 := '17702161820113', [3].QAD := '607020', [3].Peso_Real := 793.0, [3].Peso_Teorico := 786.0, [3].No_Cajas := 48, [3].Consec := 4, [3].Envase := 17250, [3].Envases_x_Caja := 1, [3].Densidad_Medida := 0.9148, [3].Linea := 5, [4].Fecha.year := 2021, [4].Fecha.Mes := 5, [4].Fecha.Dia := 27, [4].Fecha.Hora := 8, [4].Fecha.Minuto := 28, [4].Fecha.Segundo := 44, [4].Fecha.Milisegundos := 653847, [4].Lote := 147, [4].Operador := 6, [4].Descripcion := 'Aceite Vegetal Torino  Exp.', [4].EAN14 := '17702161820113', [4].QAD := '607020', [4].Peso_Real := 792.0, [4].Peso_Teorico := 786.0, [4].No_Cajas := 48, [4].Consec := 5, [4].Envase := 17250, [4].Envases_x_Caja := 1, [4].Densidad_Medida := 0.9148, [4].Linea := 5, [5].Fecha.year := 2021, [5].Fecha.Mes := 5, [5].Fecha.Dia := 27, [5].Fecha.Hora := 8, [5].Fecha.Minuto := 32, [5].Fecha.Segundo := 26, [5].Fecha.Milisegundos := 274275, [5].Lote := 147, [5].Operador := 6, [5].Descripcion := 'Aceite Vegetal Torino  Exp.', [5].EAN14 := '17702161820113', [5].QAD := '607020', [5].Peso_Real := 790.0, [5].Peso_Teorico := 786.0, [5].No_Cajas := 48, [5].Consec := 6, [5].Envase := 17250, [5].Envases_x_Caja := 1, [5].Densidad_Medida := 0.9148, [5].Linea := 5,
        [6].Fecha.year := 2021, [6].Fecha.Mes := 5, [6].Fecha.Dia := 27, [6].Fecha.Hora := 8, [6].Fecha.Minuto := 37, [6].Fecha.Segundo := 37, [6].Fecha.Milisegundos := 41030, [6].Lote := 147, [6].Operador := 6, [6].Descripcion := 'Aceite Vegetal Torino  Exp.', [6].EAN14 := '17702161820113', [6].QAD := '607020', [6].Peso_Real := 789.0, [6].Peso_Teorico := 786.0, [6].No_Cajas := 48, [6].Consec := 7, [6].Envase := 17250, [6].Envases_x_Caja := 1, [6].Densidad_Medida := 0.9148, [6].Linea := 5, [7].Fecha.year := 2021, [7].Fecha.Mes := 5, [7].Fecha.Dia := 27, [7].Fecha.Hora := 8, [7].Fecha.Minuto := 41, [7].Fecha.Segundo := 34, [7].Fecha.Milisegundos := 580309, [7].Lote := 147, [7].Operador := 6, [7].Descripcion := 'Aceite Vegetal Torino  Exp.', [7].EAN14 := '17702161820113', [7].QAD := '607020', [7].Peso_Real := 787.0, [7].Peso_Teorico := 786.0, [7].No_Cajas := 48, [7].Consec := 8, [7].Envase := 17250, [7].Envases_x_Caja := 1, [7].Densidad_Medida := 0.9148, [7].Linea := 5, [8].Fecha.year := 2021, [8].Fecha.Mes := 5, [8].Fecha.Dia := 27, [8].Fecha.Hora := 8, [8].Fecha.Minuto := 45, [8].Fecha.Segundo := 42, [8].Fecha.Milisegundos := 193421, [8].Lote := 147, [8].Operador := 6, [8].Descripcion := 'Aceite Vegetal Torino  Exp.', [8].EAN14 := '17702161820113', [8].QAD := '607020', [8].Peso_Real := 788.0, [8].Peso_Teorico := 786.0, [8].No_Cajas := 48, [8].Consec := 9, [8].Envase := 17250, [8].Envases_x_Caja := 1, [8].Densidad_Medida := 0.9148, [8].Linea := 5,
        [9].Fecha.year := 2021, [9].Fecha.Mes := 5, [9].Fecha.Dia := 27, [9].Fecha.Hora := 8, [9].Fecha.Minuto := 49, [9].Fecha.Segundo := 12, [9].Fecha.Milisegundos := 484924, [9].Lote := 147, [9].Operador := 6, [9].Descripcion := 'Aceite Vegetal Torino  Exp.', [9].EAN14 := '17702161820113', [9].QAD := '607020', [9].Peso_Real := 787.0, [9].Peso_Teorico := 786.0, [9].No_Cajas := 48, [9].Consec := 10, [9].Envase := 17250, [9].Envases_x_Caja := 1, [9].Densidad_Medida := 0.9148, [9].Linea := 5, [10].Fecha.year := 2021, [10].Fecha.Mes := 5, [10].Fecha.Dia := 27, [10].Fecha.Hora := 9, [10].Fecha.Minuto := 3, [10].Fecha.Segundo := 17, [10].Fecha.Milisegundos := 455799, [10].Lote := 147, [10].Operador := 6, [10].Descripcion := 'Aceite Vegetal Torino  Exp.', [10].EAN14 := '17702161820113', [10].QAD := '607020', [10].Peso_Real := 789.0, [10].Peso_Teorico := 786.0, [10].No_Cajas := 48, [10].Consec := 11, [10].Envase := 17250, [10].Envases_x_Caja := 1, [10].Densidad_Medida := 0.9148, [10].Linea := 5, [11].Fecha.year := 2021, [11].Fecha.Mes := 5, [11].Fecha.Dia := 27, [11].Fecha.Hora := 9, [11].Fecha.Minuto := 8, [11].Fecha.Segundo := 26, [11].Fecha.Milisegundos := 246092, [11].Lote := 147, [11].Operador := 6, [11].Descripcion := 'Aceite Vegetal Torino  Exp.', [11].EAN14 := '17702161820113', [11].QAD := '607020', [11].Peso_Real := 792.0, [11].Peso_Teorico := 786.0, [11].No_Cajas := 48, [11].Consec := 12, [11].Envase := 17250, [11].Envases_x_Caja := 1, [11].Densidad_Medida := 0.9148, [11].Linea := 5,
        [12].Fecha.year := 2021, [12].Fecha.Mes := 5, [12].Fecha.Dia := 27, [12].Fecha.Hora := 9, [12].Fecha.Minuto := 16, [12].Fecha.Segundo := 47, [12].Fecha.Milisegundos := 114605, [12].Lote := 147, [12].Operador := 6, [12].Descripcion := 'Aceite Vegetal Torino  Exp.', [12].EAN14 := '17702161820113', [12].QAD := '607020', [12].Peso_Real := 789.0, [12].Peso_Teorico := 786.0, [12].No_Cajas := 48, [12].Consec := 14, [12].Envase := 17250, [12].Envases_x_Caja := 1, [12].Densidad_Medida := 0.9148, [12].Linea := 5, [13].Fecha.year := 2021, [13].Fecha.Mes := 5, [13].Fecha.Dia := 27, [13].Fecha.Hora := 9, [13].Fecha.Minuto := 20, [13].Fecha.Segundo := 49, [13].Fecha.Milisegundos := 264386, [13].Lote := 147, [13].Operador := 6, [13].Descripcion := 'Aceite Vegetal Torino  Exp.', [13].EAN14 := '17702161820113', [13].QAD := '607020', [13].Peso_Real := 788.0, [13].Peso_Teorico := 786.0, [13].No_Cajas := 48, [13].Consec := 15, [13].Envase := 17250, [13].Envases_x_Caja := 1, [13].Densidad_Medida := 0.9148, [13].Linea := 5, [14].Fecha.year := 2021, [14].Fecha.Mes := 5, [14].Fecha.Dia := 27, [14].Fecha.Hora := 9, [14].Fecha.Minuto := 24, [14].Fecha.Segundo := 48, [14].Fecha.Milisegundos := 961089, [14].Lote := 147, [14].Operador := 6, [14].Descripcion := 'Aceite Vegetal Torino  Exp.', [14].EAN14 := '17702161820113', [14].QAD := '607020', [14].Peso_Real := 789.0, [14].Peso_Teorico := 786.0, [14].No_Cajas := 48, [14].Consec := 16, [14].Envase := 17250, [14].Envases_x_Caja := 1, [14].Densidad_Medida := 0.9148, [14].Linea := 5,
        [15].Fecha.year := 2021, [15].Fecha.Mes := 5, [15].Fecha.Dia := 27, [15].Fecha.Hora := 9, [15].Fecha.Minuto := 28, [15].Fecha.Segundo := 40, [15].Fecha.Milisegundos := 76249, [15].Lote := 147, [15].Operador := 6, [15].Descripcion := 'Aceite Vegetal Torino  Exp.', [15].EAN14 := '17702161820113', [15].QAD := '607020', [15].Peso_Real := 789.0, [15].Peso_Teorico := 786.0, [15].No_Cajas := 48, [15].Consec := 18, [15].Envase := 17250, [15].Envases_x_Caja := 1, [15].Densidad_Medida := 0.9148, [15].Linea := 5, [16].Fecha.year := 2021, [16].Fecha.Mes := 5, [16].Fecha.Dia := 27, [16].Fecha.Hora := 9, [16].Fecha.Minuto := 33, [16].Fecha.Segundo := 54, [16].Fecha.Milisegundos := 659162, [16].Lote := 147, [16].Operador := 6, [16].Descripcion := 'Aceite Vegetal Torino  Exp.', [16].EAN14 := '17702161820113', [16].QAD := '607020', [16].Peso_Real := 785.0, [16].Peso_Teorico := 786.0, [16].No_Cajas := 48, [16].Consec := 20, [16].Envase := 17250, [16].Envases_x_Caja := 1, [16].Densidad_Medida := 0.9148, [16].Linea := 5, [17].Fecha.year := 2021, [17].Fecha.Mes := 5, [17].Fecha.Dia := 27, [17].Fecha.Hora := 9, [17].Fecha.Minuto := 38, [17].Fecha.Segundo := 48, [17].Fecha.Milisegundos := 510874, [17].Lote := 147, [17].Operador := 6, [17].Descripcion := 'Aceite Vegetal Torino  Exp.', [17].EAN14 := '17702161820113', [17].QAD := '607020', [17].Peso_Real := 788.0, [17].Peso_Teorico := 786.0, [17].No_Cajas := 48, [17].Consec := 21, [17].Envase := 17250, [17].Envases_x_Caja := 1, [17].Densidad_Medida := 0.9148, [17].Linea := 5,
        [18].Fecha.year := 2021, [18].Fecha.Mes := 5, [18].Fecha.Dia := 27, [18].Fecha.Hora := 9, [18].Fecha.Minuto := 42, [18].Fecha.Segundo := 43, [18].Fecha.Milisegundos := 692690, [18].Lote := 147, [18].Operador := 6, [18].Descripcion := 'Aceite Vegetal Torino  Exp.', [18].EAN14 := '17702161820113', [18].QAD := '607020', [18].Peso_Real := 788.0, [18].Peso_Teorico := 786.0, [18].No_Cajas := 48, [18].Consec := 22, [18].Envase := 17250, [18].Envases_x_Caja := 1, [18].Densidad_Medida := 0.9148, [18].Linea := 5, [19].Fecha.year := 2021, [19].Fecha.Mes := 5, [19].Fecha.Dia := 27, [19].Fecha.Hora := 9, [19].Fecha.Minuto := 47, [19].Fecha.Segundo := 11, [19].Fecha.Milisegundos := 196960, [19].Lote := 147, [19].Operador := 6, [19].Descripcion := 'Aceite Vegetal Torino  Exp.', [19].EAN14 := '17702161820113', [19].QAD := '607020', [19].Peso_Real := 788.0, [19].Peso_Teorico := 786.0, [19].No_Cajas := 48, [19].Consec := 24, [19].Envase := 17250, [19].Envases_x_Caja := 1, [19].Densidad_Medida := 0.9148, [19].Linea := 5, [20].Fecha.year := 2021, [20].Fecha.Mes := 5, [20].Fecha.Dia := 27, [20].Fecha.Hora := 9, [20].Fecha.Minuto := 52, [20].Fecha.Segundo := 45, [20].Fecha.Milisegundos := 491531, [20].Lote := 147, [20].Operador := 6, [20].Descripcion := 'Aceite Vegetal Torino  Exp.', [20].EAN14 := '17702161820113', [20].QAD := '607020', [20].Peso_Real := 788.0, [20].Peso_Teorico := 786.0, [20].No_Cajas := 48, [20].Consec := 26, [20].Envase := 17250, [20].Envases_x_Caja := 1, [20].Densidad_Medida := 0.9148, [20].Linea := 5,
        [21].Fecha.year := 2021, [21].Fecha.Mes := 5, [21].Fecha.Dia := 27, [21].Fecha.Hora := 9, [21].Fecha.Minuto := 58, [21].Fecha.Segundo := 30, [21].Fecha.Milisegundos := 407702, [21].Lote := 147, [21].Operador := 6, [21].Descripcion := 'Aceite Vegetal Torino  Exp.', [21].EAN14 := '17702161820113', [21].QAD := '607020', [21].Peso_Real := 790.0, [21].Peso_Teorico := 786.0, [21].No_Cajas := 48, [21].Consec := 27, [21].Envase := 17250, [21].Envases_x_Caja := 1, [21].Densidad_Medida := 0.9148, [21].Linea := 5, [22].Fecha.year := 2021, [22].Fecha.Mes := 5, [22].Fecha.Dia := 27, [22].Fecha.Hora := 10, [22].Fecha.Minuto := 3, [22].Fecha.Segundo := 52, [22].Fecha.Milisegundos := 388294, [22].Lote := 147, [22].Operador := 6, [22].Descripcion := 'Aceite Vegetal Torino  Exp.', [22].EAN14 := '17702161820113', [22].QAD := '607020', [22].Peso_Real := 790.0, [22].Peso_Teorico := 786.0, [22].No_Cajas := 48, [22].Consec := 28, [22].Envase := 17250, [22].Envases_x_Caja := 1, [22].Densidad_Medida := 0.9148, [22].Linea := 5, [23].Fecha.year := 2021, [23].Fecha.Mes := 5, [23].Fecha.Dia := 27, [23].Fecha.Hora := 10, [23].Fecha.Minuto := 17, [23].Fecha.Segundo := 7, [23].Fecha.Milisegundos := 441628, [23].Lote := 147, [23].Operador := 6, [23].Descripcion := 'Aceite Vegetal Torino  Exp.', [23].EAN14 := '17702161820113', [23].QAD := '607020', [23].Peso_Real := 790.0, [23].Peso_Teorico := 786.0, [23].No_Cajas := 48, [23].Consec := 29, [23].Envase := 17250, [23].Envases_x_Caja := 1, [23].Densidad_Medida := 0.9148, [23].Linea := 5,
        [24].Fecha.year := 2021, [24].Fecha.Mes := 5, [24].Fecha.Dia := 27, [24].Fecha.Hora := 10, [24].Fecha.Minuto := 21, [24].Fecha.Segundo := 17, [24].Fecha.Milisegundos := 311569, [24].Lote := 147, [24].Operador := 6, [24].Descripcion := 'Aceite Vegetal Torino  Exp.', [24].EAN14 := '17702161820113', [24].QAD := '607020', [24].Peso_Real := 792.0, [24].Peso_Teorico := 786.0, [24].No_Cajas := 48, [24].Consec := 30, [24].Envase := 17250, [24].Envases_x_Caja := 1, [24].Densidad_Medida := 0.9148, [24].Linea := 5, [25].Fecha.year := 2021, [25].Fecha.Mes := 5, [25].Fecha.Dia := 27, [25].Fecha.Hora := 10, [25].Fecha.Minuto := 25, [25].Fecha.Segundo := 29, [25].Fecha.Milisegundos := 60847, [25].Lote := 147, [25].Operador := 6, [25].Descripcion := 'Aceite Vegetal Torino  Exp.', [25].EAN14 := '17702161820113', [25].QAD := '607020', [25].Peso_Real := 789.0, [25].Peso_Teorico := 786.0, [25].No_Cajas := 48, [25].Consec := 31, [25].Envase := 17250, [25].Envases_x_Caja := 1, [25].Densidad_Medida := 0.9148, [25].Linea := 5, [26].Fecha.year := 2021, [26].Fecha.Mes := 5, [26].Fecha.Dia := 27, [26].Fecha.Hora := 11, [26].Fecha.Minuto := 14, [26].Fecha.Segundo := 30, [26].Fecha.Milisegundos := 310820, [26].Lote := 147, [26].Operador := 6, [26].Descripcion := 'Aceite Vegetal Torino  Exp.', [26].EAN14 := '17702161820113', [26].QAD := '607020', [26].Peso_Real := 789.0, [26].Peso_Teorico := 786.0, [26].No_Cajas := 48, [26].Consec := 39, [26].Envase := 17250, [26].Envases_x_Caja := 1, [26].Densidad_Medida := 0.9148, [26].Linea := 5,
        [27].Fecha.year := 2021, [27].Fecha.Mes := 5, [27].Fecha.Dia := 27, [27].Fecha.Hora := 11, [27].Fecha.Minuto := 29, [27].Fecha.Segundo := 2, [27].Fecha.Milisegundos := 929977, [27].Lote := 147, [27].Operador := 6, [27].Descripcion := 'Aceite Vegetal Torino  Exp.', [27].EAN14 := '17702161820113', [27].QAD := '607020', [27].Peso_Real := 785.0, [27].Peso_Teorico := 786.0, [27].No_Cajas := 48, [27].Consec := 41, [27].Envase := 17250, [27].Envases_x_Caja := 1, [27].Densidad_Medida := 0.9148, [27].Linea := 5, [28].Fecha.year := 2021, [28].Fecha.Mes := 5, [28].Fecha.Dia := 27, [28].Fecha.Hora := 11, [28].Fecha.Minuto := 35, [28].Fecha.Segundo := 18, [28].Fecha.Milisegundos := 824860, [28].Lote := 147, [28].Operador := 6, [28].Descripcion := 'Aceite Vegetal Torino  Exp.', [28].EAN14 := '17702161820113', [28].QAD := '607020', [28].Peso_Real := 788.0, [28].Peso_Teorico := 786.0, [28].No_Cajas := 48, [28].Consec := 43, [28].Envase := 17250, [28].Envases_x_Caja := 1, [28].Densidad_Medida := 0.9148, [28].Linea := 5, [29].Fecha.year := 2021, [29].Fecha.Mes := 5, [29].Fecha.Dia := 27, [29].Fecha.Hora := 11, [29].Fecha.Minuto := 42, [29].Fecha.Segundo := 29, [29].Fecha.Milisegundos := 931870, [29].Lote := 147, [29].Operador := 6, [29].Descripcion := 'Aceite Vegetal Torino  Exp.', [29].EAN14 := '17702161820113', [29].QAD := '607020', [29].Peso_Real := 788.0, [29].Peso_Teorico := 786.0, [29].No_Cajas := 48, [29].Consec := 46, [29].Envase := 17250, [29].Envases_x_Caja := 1, [29].Densidad_Medida := 0.9148, [29].Linea := 5,
        [30].Fecha.year := 2021, [30].Fecha.Mes := 5, [30].Fecha.Dia := 27, [30].Fecha.Hora := 11, [30].Fecha.Minuto := 48, [30].Fecha.Segundo := 14, [30].Fecha.Milisegundos := 984158, [30].Lote := 147, [30].Operador := 6, [30].Descripcion := 'Aceite Vegetal Torino  Exp.', [30].EAN14 := '17702161820113', [30].QAD := '607020', [30].Peso_Real := 788.0, [30].Peso_Teorico := 786.0, [30].No_Cajas := 48, [30].Consec := 49, [30].Envase := 17250, [30].Envases_x_Caja := 1, [30].Densidad_Medida := 0.9148, [30].Linea := 5, [31].Fecha.year := 2021, [31].Fecha.Mes := 5, [31].Fecha.Dia := 27, [31].Fecha.Hora := 11, [31].Fecha.Minuto := 51, [31].Fecha.Segundo := 55, [31].Fecha.Milisegundos := 864354, [31].Lote := 147, [31].Operador := 6, [31].Descripcion := 'Aceite Vegetal Torino  Exp.', [31].EAN14 := '17702161820113', [31].QAD := '607020', [31].Peso_Real := 785.0, [31].Peso_Teorico := 786.0, [31].No_Cajas := 48, [31].Consec := 51, [31].Envase := 17250, [31].Envases_x_Caja := 1, [31].Densidad_Medida := 0.9148, [31].Linea := 5, [32].Fecha.year := 2021, [32].Fecha.Mes := 5, [32].Fecha.Dia := 27, [32].Fecha.Hora := 11, [32].Fecha.Minuto := 58, [32].Fecha.Segundo := 24, [32].Fecha.Milisegundos := 43089, [32].Lote := 147, [32].Operador := 6, [32].Descripcion := 'Aceite Vegetal Torino  Exp.', [32].EAN14 := '17702161820113', [32].QAD := '607020', [32].Peso_Real := 788.0, [32].Peso_Teorico := 786.0, [32].No_Cajas := 48, [32].Consec := 53, [32].Envase := 17250, [32].Envases_x_Caja := 1, [32].Densidad_Medida := 0.9148, [32].Linea := 5,
        [33].Fecha.year := 2021, [33].Fecha.Mes := 5, [33].Fecha.Dia := 27, [33].Fecha.Hora := 12, [33].Fecha.Minuto := 3, [33].Fecha.Segundo := 6, [33].Fecha.Milisegundos := 147319, [33].Lote := 147, [33].Operador := 6, [33].Descripcion := 'Aceite Vegetal Torino  Exp.', [33].EAN14 := '17702161820113', [33].QAD := '607020', [33].Peso_Real := 790.0, [33].Peso_Teorico := 786.0, [33].No_Cajas := 48, [33].Consec := 54, [33].Envase := 17250, [33].Envases_x_Caja := 1, [33].Densidad_Medida := 0.9148, [33].Linea := 5, [34].Fecha.year := 2021, [34].Fecha.Mes := 5, [34].Fecha.Dia := 27, [34].Fecha.Hora := 12, [34].Fecha.Minuto := 7, [34].Fecha.Segundo := 40, [34].Fecha.Milisegundos := 542686, [34].Lote := 147, [34].Operador := 6, [34].Descripcion := 'Aceite Vegetal Torino  Exp.', [34].EAN14 := '17702161820113', [34].QAD := '607020', [34].Peso_Real := 790.0, [34].Peso_Teorico := 786.0, [34].No_Cajas := 48, [34].Consec := 56, [34].Envase := 17250, [34].Envases_x_Caja := 1, [34].Densidad_Medida := 0.9148, [34].Linea := 5, [35].Fecha.year := 2021, [35].Fecha.Mes := 5, [35].Fecha.Dia := 27, [35].Fecha.Hora := 12, [35].Fecha.Minuto := 12, [35].Fecha.Segundo := 29, [35].Fecha.Milisegundos := 877264, [35].Lote := 147, [35].Operador := 6, [35].Descripcion := 'Aceite Vegetal Torino  Exp.', [35].EAN14 := '17702161820113', [35].QAD := '607020', [35].Peso_Real := 788.0, [35].Peso_Teorico := 786.0, [35].No_Cajas := 48, [35].Consec := 59, [35].Envase := 17250, [35].Envases_x_Caja := 1, [35].Densidad_Medida := 0.9148, [35].Linea := 5,
        [36].Fecha.year := 2021, [36].Fecha.Mes := 5, [36].Fecha.Dia := 27, [36].Fecha.Hora := 12, [36].Fecha.Minuto := 16, [36].Fecha.Segundo := 33, [36].Fecha.Milisegundos := 977790, [36].Lote := 147, [36].Operador := 6, [36].Descripcion := 'Aceite Vegetal Torino  Exp.', [36].EAN14 := '17702161820113', [36].QAD := '607020', [36].Peso_Real := 790.0, [36].Peso_Teorico := 786.0, [36].No_Cajas := 48, [36].Consec := 61, [36].Envase := 17250, [36].Envases_x_Caja := 1, [36].Densidad_Medida := 0.9148, [36].Linea := 5, [37].Fecha.year := 2021, [37].Fecha.Mes := 5, [37].Fecha.Dia := 27, [37].Fecha.Hora := 12, [37].Fecha.Minuto := 22, [37].Fecha.Segundo := 52, [37].Fecha.Milisegundos := 436140, [37].Lote := 147, [37].Operador := 6, [37].Descripcion := 'Aceite Vegetal Torino  Exp.', [37].EAN14 := '17702161820113', [37].QAD := '607020', [37].Peso_Real := 787.0, [37].Peso_Teorico := 786.0, [37].No_Cajas := 48, [37].Consec := 63, [37].Envase := 17250, [37].Envases_x_Caja := 1, [37].Densidad_Medida := 0.9148, [37].Linea := 5, [38].Fecha.year := 2021, [38].Fecha.Mes := 5, [38].Fecha.Dia := 27, [38].Fecha.Hora := 12, [38].Fecha.Minuto := 23, [38].Fecha.Segundo := 48, [38].Fecha.Milisegundos := 375656, [38].Lote := 147, [38].Operador := 6, [38].Descripcion := 'Aceite Vegetal Torino  Exp.', [38].EAN14 := '17702161820113', [38].QAD := '607020', [38].Peso_Real := 787.0, [38].Peso_Teorico := 786.0, [38].No_Cajas := 48, [38].Consec := 65, [38].Envase := 17250, [38].Envases_x_Caja := 1, [38].Densidad_Medida := 0.9148, [38].Linea := 5,
        [39].Fecha.year := 2021, [39].Fecha.Mes := 5, [39].Fecha.Dia := 27, [39].Fecha.Hora := 12, [39].Fecha.Minuto := 27, [39].Fecha.Segundo := 6, [39].Fecha.Milisegundos := 918617, [39].Lote := 147, [39].Operador := 6, [39].Descripcion := 'Aceite Vegetal Torino  Exp.', [39].EAN14 := '17702161820113', [39].QAD := '607020', [39].Peso_Real := 814.0, [39].Peso_Teorico := 786.0, [39].No_Cajas := 48, [39].Consec := 66, [39].Envase := 17250, [39].Envases_x_Caja := 1, [39].Densidad_Medida := 0.9148, [39].Linea := 5, [40].Fecha.year := 2021, [40].Fecha.Mes := 5, [40].Fecha.Dia := 27, [40].Fecha.Hora := 12, [40].Fecha.Minuto := 30, [40].Fecha.Segundo := 31, [40].Fecha.Milisegundos := 970846, [40].Lote := 147, [40].Operador := 6, [40].Descripcion := 'Aceite Vegetal Torino  Exp.', [40].EAN14 := '17702161820113', [40].QAD := '607020', [40].Peso_Real := 789.0, [40].Peso_Teorico := 786.0, [40].No_Cajas := 48, [40].Consec := 67, [40].Envase := 17250, [40].Envases_x_Caja := 1, [40].Densidad_Medida := 0.9148, [40].Linea := 5, [41].Fecha.year := 2021, [41].Fecha.Mes := 5, [41].Fecha.Dia := 27, [41].Fecha.Hora := 12, [41].Fecha.Minuto := 34, [41].Fecha.Segundo := 5, [41].Fecha.Milisegundos := 792914, [41].Lote := 147, [41].Operador := 6, [41].Descripcion := 'Aceite Vegetal Torino  Exp.', [41].EAN14 := '17702161820113', [41].QAD := '607020', [41].Peso_Real := 788.0, [41].Peso_Teorico := 786.0, [41].No_Cajas := 48, [41].Consec := 69, [41].Envase := 17250, [41].Envases_x_Caja := 1, [41].Densidad_Medida := 0.9148, [41].Linea := 5,
        [42].Fecha.year := 2021, [42].Fecha.Mes := 5, [42].Fecha.Dia := 27, [42].Fecha.Hora := 12, [42].Fecha.Minuto := 38, [42].Fecha.Segundo := 13, [42].Fecha.Milisegundos := 633087, [42].Lote := 147, [42].Operador := 6, [42].Descripcion := 'Aceite Vegetal Torino  Exp.', [42].EAN14 := '17702161820113', [42].QAD := '607020', [42].Peso_Real := 742.0, [42].Peso_Teorico := 786.0, [42].No_Cajas := 48, [42].Consec := 71, [42].Envase := 17250, [42].Envases_x_Caja := 1, [42].Densidad_Medida := 0.9148, [42].Linea := 5, [43].Fecha.year := 2021, [43].Fecha.Mes := 5, [43].Fecha.Dia := 27, [43].Fecha.Hora := 12, [43].Fecha.Minuto := 45, [43].Fecha.Segundo := 17, [43].Fecha.Milisegundos := 629727, [43].Lote := 147, [43].Operador := 6, [43].Descripcion := 'Aceite Vegetal Torino  Exp.', [43].EAN14 := '17702161820113', [43].QAD := '607020', [43].Peso_Real := 789.0, [43].Peso_Teorico := 786.0, [43].No_Cajas := 48, [43].Consec := 74, [43].Envase := 17250, [43].Envases_x_Caja := 1, [43].Densidad_Medida := 0.9148, [43].Linea := 5, [44].Fecha.year := 2021, [44].Fecha.Mes := 5, [44].Fecha.Dia := 27, [44].Fecha.Hora := 12, [44].Fecha.Minuto := 49, [44].Fecha.Segundo := 49, [44].Fecha.Milisegundos := 292109, [44].Lote := 147, [44].Operador := 6, [44].Descripcion := 'Aceite Vegetal Torino  Exp.', [44].EAN14 := '17702161820113', [44].QAD := '607020', [44].Peso_Real := 788.0, [44].Peso_Teorico := 786.0, [44].No_Cajas := 48, [44].Consec := 77, [44].Envase := 17250, [44].Envases_x_Caja := 1, [44].Densidad_Medida := 0.9148, [44].Linea := 5,
        [45].Fecha.year := 2021, [45].Fecha.Mes := 5, [45].Fecha.Dia := 27, [45].Fecha.Hora := 12, [45].Fecha.Minuto := 54, [45].Fecha.Segundo := 45, [45].Fecha.Milisegundos := 664920, [45].Lote := 147, [45].Operador := 6, [45].Descripcion := 'Aceite Vegetal Torino  Exp.', [45].EAN14 := '17702161820113', [45].QAD := '607020', [45].Peso_Real := 788.0, [45].Peso_Teorico := 786.0, [45].No_Cajas := 48, [45].Consec := 80, [45].Envase := 17250, [45].Envases_x_Caja := 1, [45].Densidad_Medida := 0.9148, [45].Linea := 5, [46].Fecha.year := 2021, [46].Fecha.Mes := 5, [46].Fecha.Dia := 27, [46].Fecha.Hora := 12, [46].Fecha.Minuto := 59, [46].Fecha.Segundo := 46, [46].Fecha.Milisegundos := 913760, [46].Lote := 147, [46].Operador := 6, [46].Descripcion := 'Aceite Vegetal Torino  Exp.', [46].EAN14 := '17702161820113', [46].QAD := '607020', [46].Peso_Real := 787.0, [46].Peso_Teorico := 786.0, [46].No_Cajas := 48, [46].Consec := 82, [46].Envase := 17250, [46].Envases_x_Caja := 1, [46].Densidad_Medida := 0.9148, [46].Linea := 5, [47].Fecha.year := 2021, [47].Fecha.Mes := 5, [47].Fecha.Dia := 27, [47].Fecha.Hora := 13, [47].Fecha.Minuto := 4, [47].Fecha.Segundo := 32, [47].Fecha.Milisegundos := 629070, [47].Lote := 147, [47].Operador := 6, [47].Descripcion := 'Aceite Vegetal Torino  Exp.', [47].EAN14 := '17702161820113', [47].QAD := '607020', [47].Peso_Real := 789.0, [47].Peso_Teorico := 786.0, [47].No_Cajas := 48, [47].Consec := 85, [47].Envase := 17250, [47].Envases_x_Caja := 1, [47].Densidad_Medida := 0.9148, [47].Linea := 5,
        [48].Fecha.year := 2021, [48].Fecha.Mes := 5, [48].Fecha.Dia := 27, [48].Fecha.Hora := 13, [48].Fecha.Minuto := 12, [48].Fecha.Segundo := 31, [48].Fecha.Milisegundos := 127420, [48].Lote := 147, [48].Operador := 6, [48].Descripcion := 'Aceite Vegetal Torino  Exp.', [48].EAN14 := '17702161820113', [48].QAD := '607020', [48].Peso_Real := 793.0, [48].Peso_Teorico := 786.0, [48].No_Cajas := 48, [48].Consec := 89, [48].Envase := 17250, [48].Envases_x_Caja := 1, [48].Densidad_Medida := 0.9148, [48].Linea := 5, [49].Fecha.year := 2021, [49].Fecha.Mes := 5, [49].Fecha.Dia := 27, [49].Fecha.Hora := 13, [49].Fecha.Minuto := 17, [49].Fecha.Segundo := 16, [49].Fecha.Milisegundos := 299229, [49].Lote := 147, [49].Operador := 6, [49].Descripcion := 'Aceite Vegetal Torino  Exp.', [49].EAN14 := '17702161820113', [49].QAD := '607020', [49].Peso_Real := 788.0, [49].Peso_Teorico := 786.0, [49].No_Cajas := 48, [49].Consec := 91, [49].Envase := 17250, [49].Envases_x_Caja := 1, [49].Densidad_Medida := 0.9148, [49].Linea := 5, [50].Fecha.year := 2021, [50].Fecha.Mes := 5, [50].Fecha.Dia := 27, [50].Fecha.Hora := 13, [50].Fecha.Minuto := 20, [50].Fecha.Segundo := 43, [50].Fecha.Milisegundos := 81946, [50].Lote := 147, [50].Operador := 6, [50].Descripcion := 'Aceite Vegetal Torino  Exp.', [50].EAN14 := '17702161820113', [50].QAD := '607020', [50].Peso_Real := 792.0, [50].Peso_Teorico := 786.0, [50].No_Cajas := 48, [50].Consec := 93, [50].Envase := 17250, [50].Envases_x_Caja := 1, [50].Densidad_Medida := 0.9148, [50].Linea := 5,
        [51].Fecha.year := 2021, [51].Fecha.Mes := 5, [51].Fecha.Dia := 27, [51].Fecha.Hora := 13, [51].Fecha.Minuto := 24, [51].Fecha.Segundo := 46, [51].Fecha.Milisegundos := 552036, [51].Lote := 147, [51].Operador := 6, [51].Descripcion := 'Aceite Vegetal Torino  Exp.', [51].EAN14 := '17702161820113', [51].QAD := '607020', [51].Peso_Real := 793.0, [51].Peso_Teorico := 786.0, [51].No_Cajas := 48, [51].Consec := 96, [51].Envase := 17250, [51].Envases_x_Caja := 1, [51].Densidad_Medida := 0.9148, [51].Linea := 5, [52].Fecha.year := 2021, [52].Fecha.Mes := 5, [52].Fecha.Dia := 27, [52].Fecha.Hora := 13, [52].Fecha.Minuto := 28, [52].Fecha.Segundo := 18, [52].Fecha.Milisegundos := 718753, [52].Lote := 147, [52].Operador := 6, [52].Descripcion := 'Aceite Vegetal Torino  Exp.', [52].EAN14 := '17702161820113', [52].QAD := '607020', [52].Peso_Real := 793.0, [52].Peso_Teorico := 786.0, [52].No_Cajas := 48, [52].Consec := 98, [52].Envase := 17250, [52].Envases_x_Caja := 1, [52].Densidad_Medida := 0.9148, [52].Linea := 5, [53].Fecha.year := 2021, [53].Fecha.Mes := 5, [53].Fecha.Dia := 27, [53].Fecha.Hora := 13, [53].Fecha.Minuto := 34, [53].Fecha.Segundo := 33, [53].Fecha.Milisegundos := 396020, [53].Lote := 147, [53].Operador := 6, [53].Descripcion := 'Aceite Vegetal Torino  Exp.', [53].EAN14 := '17702161820113', [53].QAD := '607020', [53].Peso_Real := 787.0, [53].Peso_Teorico := 786.0, [53].No_Cajas := 48, [53].Consec := 101, [53].Envase := 17250, [53].Envases_x_Caja := 1, [53].Densidad_Medida := 0.9148, [53].Linea := 5,
        [54].Fecha.year := 2021, [54].Fecha.Mes := 5, [54].Fecha.Dia := 27, [54].Fecha.Hora := 13, [54].Fecha.Minuto := 38, [54].Fecha.Segundo := 50, [54].Fecha.Milisegundos := 151717, [54].Lote := 147, [54].Operador := 6, [54].Descripcion := 'Aceite Vegetal Torino  Exp.', [54].EAN14 := '17702161820113', [54].QAD := '607020', [54].Peso_Real := 787.0, [54].Peso_Teorico := 786.0, [54].No_Cajas := 48, [54].Consec := 104, [54].Envase := 17250, [54].Envases_x_Caja := 1, [54].Densidad_Medida := 0.9148, [54].Linea := 5, [55].Fecha.year := 2021, [55].Fecha.Mes := 5, [55].Fecha.Dia := 27, [55].Fecha.Hora := 13, [55].Fecha.Minuto := 43, [55].Fecha.Segundo := 38, [55].Fecha.Milisegundos := 38315, [55].Lote := 147, [55].Operador := 6, [55].Descripcion := 'Aceite Vegetal Torino  Exp.', [55].EAN14 := '17702161820113', [55].QAD := '607020', [55].Peso_Real := 788.0, [55].Peso_Teorico := 786.0, [55].No_Cajas := 48, [55].Consec := 107, [55].Envase := 17250, [55].Envases_x_Caja := 1, [55].Densidad_Medida := 0.9148, [55].Linea := 5, [56].Fecha.year := 2021, [56].Fecha.Mes := 5, [56].Fecha.Dia := 27, [56].Fecha.Hora := 13, [56].Fecha.Minuto := 48, [56].Fecha.Segundo := 11, [56].Fecha.Milisegundos := 485018, [56].Lote := 147, [56].Operador := 6, [56].Descripcion := 'Aceite Vegetal Torino  Exp.', [56].EAN14 := '17702161820113', [56].QAD := '607020', [56].Peso_Real := 789.0, [56].Peso_Teorico := 786.0, [56].No_Cajas := 48, [56].Consec := 109, [56].Envase := 17250, [56].Envases_x_Caja := 1, [56].Densidad_Medida := 0.9148, [56].Linea := 5,
        [57].Fecha.year := 2021, [57].Fecha.Mes := 5, [57].Fecha.Dia := 27, [57].Fecha.Hora := 13, [57].Fecha.Minuto := 53, [57].Fecha.Segundo := 13, [57].Fecha.Milisegundos := 883574, [57].Lote := 147, [57].Operador := 6, [57].Descripcion := 'Aceite Vegetal Torino  Exp.', [57].EAN14 := '17702161820113', [57].QAD := '607020', [57].Peso_Real := 787.0, [57].Peso_Teorico := 786.0, [57].No_Cajas := 48, [57].Consec := 112, [57].Envase := 17250, [57].Envases_x_Caja := 1, [57].Densidad_Medida := 0.9148, [57].Linea := 5, [58].Fecha.year := 2021, [58].Fecha.Mes := 5, [58].Fecha.Dia := 27, [58].Fecha.Hora := 14, [58].Fecha.Minuto := 1, [58].Fecha.Segundo := 23, [58].Fecha.Milisegundos := 845245, [58].Lote := 147, [58].Operador := 6, [58].Descripcion := 'Aceite Vegetal Torino  Exp.', [58].EAN14 := '17702161820113', [58].QAD := '607020', [58].Peso_Real := 790.0, [58].Peso_Teorico := 786.0, [58].No_Cajas := 48, [58].Consec := 116, [58].Envase := 17250, [58].Envases_x_Caja := 1, [58].Densidad_Medida := 0.9148, [58].Linea := 5, [59].Fecha.year := 2021, [59].Fecha.Mes := 5, [59].Fecha.Dia := 27, [59].Fecha.Hora := 14, [59].Fecha.Minuto := 7, [59].Fecha.Segundo := 8, [59].Fecha.Milisegundos := 597590, [59].Lote := 147, [59].Operador := 6, [59].Descripcion := 'Aceite Vegetal Torino  Exp.', [59].EAN14 := '17702161820113', [59].QAD := '607020', [59].Peso_Real := 788.0, [59].Peso_Teorico := 786.0, [59].No_Cajas := 48, [59].Consec := 118, [59].Envase := 17250, [59].Envases_x_Caja := 1, [59].Densidad_Medida := 0.9148, [59].Linea := 5,
        [60].Fecha.year := 2021, [60].Fecha.Mes := 5, [60].Fecha.Dia := 27, [60].Fecha.Hora := 14, [60].Fecha.Minuto := 11, [60].Fecha.Segundo := 36, [60].Fecha.Milisegundos := 606941, [60].Lote := 147, [60].Operador := 6, [60].Descripcion := 'Aceite Vegetal Torino  Exp.', [60].EAN14 := '17702161820113', [60].QAD := '607020', [60].Peso_Real := 784.0, [60].Peso_Teorico := 786.0, [60].No_Cajas := 48, [60].Consec := 120, [60].Envase := 17250, [60].Envases_x_Caja := 1, [60].Densidad_Medida := 0.9148, [60].Linea := 5, [61].Fecha.year := 2021, [61].Fecha.Mes := 5, [61].Fecha.Dia := 27, [61].Fecha.Hora := 14, [61].Fecha.Minuto := 16, [61].Fecha.Segundo := 40, [61].Fecha.Milisegundos := 178533, [61].Lote := 147, [61].Operador := 6, [61].Descripcion := 'Aceite Vegetal Torino  Exp.', [61].EAN14 := '17702161820113', [61].QAD := '607020', [61].Peso_Real := 794.0, [61].Peso_Teorico := 786.0, [61].No_Cajas := 48, [61].Consec := 123, [61].Envase := 17250, [61].Envases_x_Caja := 1, [61].Densidad_Medida := 0.9148, [61].Linea := 5, [62].Fecha.year := 2021, [62].Fecha.Mes := 5, [62].Fecha.Dia := 27, [62].Fecha.Hora := 14, [62].Fecha.Minuto := 24, [62].Fecha.Segundo := 37, [62].Fecha.Milisegundos := 944953, [62].Lote := 147, [62].Operador := 6, [62].Descripcion := 'Aceite Vegetal Torino  Exp.', [62].EAN14 := '17702161820113', [62].QAD := '607020', [62].Peso_Real := 788.0, [62].Peso_Teorico := 786.0, [62].No_Cajas := 48, [62].Consec := 124, [62].Envase := 17250, [62].Envases_x_Caja := 1, [62].Densidad_Medida := 0.9148, [62].Linea := 5,
        [63].Fecha.year := 2021, [63].Fecha.Mes := 5, [63].Fecha.Dia := 27, [63].Fecha.Hora := 14, [63].Fecha.Minuto := 33, [63].Fecha.Segundo := 27, [63].Fecha.Milisegundos := 894406, [63].Lote := 147, [63].Operador := 6, [63].Descripcion := 'Aceite Vegetal Torino  Exp.', [63].EAN14 := '17702161820113', [63].QAD := '607020', [63].Peso_Real := 789.0, [63].Peso_Teorico := 786.0, [63].No_Cajas := 48, [63].Consec := 125, [63].Envase := 17250, [63].Envases_x_Caja := 1, [63].Densidad_Medida := 0.9148, [63].Linea := 5, [64].Fecha.year := 2021, [64].Fecha.Mes := 5, [64].Fecha.Dia := 27, [64].Fecha.Hora := 14, [64].Fecha.Minuto := 38, [64].Fecha.Segundo := 45, [64].Fecha.Milisegundos := 262002, [64].Lote := 147, [64].Operador := 6, [64].Descripcion := 'Aceite Vegetal Torino  Exp.', [64].EAN14 := '17702161820113', [64].QAD := '607020', [64].Peso_Real := 787.0, [64].Peso_Teorico := 786.0, [64].No_Cajas := 48, [64].Consec := 126, [64].Envase := 17250, [64].Envases_x_Caja := 1, [64].Densidad_Medida := 0.9148, [64].Linea := 5, [65].Fecha.year := 2021, [65].Fecha.Mes := 5, [65].Fecha.Dia := 27, [65].Fecha.Hora := 14, [65].Fecha.Minuto := 44, [65].Fecha.Segundo := 15, [65].Fecha.Milisegundos := 380887, [65].Lote := 147, [65].Operador := 6, [65].Descripcion := 'Aceite Vegetal Torino  Exp.', [65].EAN14 := '17702161820113', [65].QAD := '607020', [65].Peso_Real := 789.0, [65].Peso_Teorico := 786.0, [65].No_Cajas := 48, [65].Consec := 127, [65].Envase := 17250, [65].Envases_x_Caja := 1, [65].Densidad_Medida := 0.9148, [65].Linea := 5,
        [66].Fecha.year := 2021, [66].Fecha.Mes := 5, [66].Fecha.Dia := 27, [66].Fecha.Hora := 14, [66].Fecha.Minuto := 49, [66].Fecha.Segundo := 59, [66].Fecha.Milisegundos := 257479, [66].Lote := 147, [66].Operador := 6, [66].Descripcion := 'Aceite Vegetal Torino  Exp.', [66].EAN14 := '17702161820113', [66].QAD := '607020', [66].Peso_Real := 788.0, [66].Peso_Teorico := 786.0, [66].No_Cajas := 48, [66].Consec := 128, [66].Envase := 17250, [66].Envases_x_Caja := 1, [66].Densidad_Medida := 0.9148, [66].Linea := 5, [67].Fecha.year := 2021, [67].Fecha.Mes := 5, [67].Fecha.Dia := 27, [67].Fecha.Hora := 14, [67].Fecha.Minuto := 54, [67].Fecha.Segundo := 56, [67].Fecha.Milisegundos := 716721, [67].Lote := 147, [67].Operador := 6, [67].Descripcion := 'Aceite Vegetal Torino  Exp.', [67].EAN14 := '17702161820113', [67].QAD := '607020', [67].Peso_Real := 789.0, [67].Peso_Teorico := 786.0, [67].No_Cajas := 48, [67].Consec := 129, [67].Envase := 17250, [67].Envases_x_Caja := 1, [67].Densidad_Medida := 0.9148, [67].Linea := 5, [68].Fecha.year := 2021, [68].Fecha.Mes := 5, [68].Fecha.Dia := 27, [68].Fecha.Hora := 15, [68].Fecha.Segundo := 21, [68].Fecha.Milisegundos := 631529, [68].Lote := 147, [68].Operador := 6, [68].Descripcion := 'Aceite Vegetal Torino  Exp.', [68].EAN14 := '17702161820113', [68].QAD := '607020', [68].Peso_Real := 789.0, [68].Peso_Teorico := 786.0, [68].No_Cajas := 48, [68].Consec := 130, [68].Envase := 17250, [68].Envases_x_Caja := 1, [68].Densidad_Medida := 0.9148, [68].Linea := 5, [69].Fecha.year := 2021,
        [69].Fecha.Mes := 5, [69].Fecha.Dia := 27, [69].Fecha.Hora := 15, [69].Fecha.Minuto := 4, [69].Fecha.Segundo := 10, [69].Fecha.Milisegundos := 704605, [69].Lote := 147, [69].Operador := 6, [69].Descripcion := 'Aceite Vegetal Torino  Exp.', [69].EAN14 := '17702161820113', [69].QAD := '607020', [69].Peso_Real := 790.0, [69].Peso_Teorico := 786.0, [69].No_Cajas := 48, [69].Consec := 131, [69].Envase := 17250, [69].Envases_x_Caja := 1, [69].Densidad_Medida := 0.9148, [69].Linea := 5, [70].Fecha.year := 2021, [70].Fecha.Mes := 5, [70].Fecha.Dia := 27, [70].Fecha.Hora := 15, [70].Fecha.Minuto := 8, [70].Fecha.Segundo := 41, [70].Fecha.Milisegundos := 219289, [70].Lote := 147, [70].Operador := 6, [70].Descripcion := 'Aceite Vegetal Torino  Exp.', [70].EAN14 := '17702161820113', [70].QAD := '607020', [70].Peso_Real := 787.0, [70].Peso_Teorico := 786.0, [70].No_Cajas := 48, [70].Consec := 132, [70].Envase := 17250, [70].Envases_x_Caja := 1, [70].Densidad_Medida := 0.9148, [70].Linea := 5, [71].Fecha.year := 2021, [71].Fecha.Mes := 5, [71].Fecha.Dia := 27, [71].Fecha.Hora := 20, [71].Fecha.Minuto := 36, [71].Fecha.Segundo := 10, [71].Fecha.Milisegundos := 90197, [71].Lote := 147, [71].Operador := 6, [71].Descripcion := 'Aceite Vegetal Torino  Exp.', [71].EAN14 := '17702161820113', [71].QAD := '607020', [71].Peso_Real := 789.0, [71].Peso_Teorico := 786.0, [71].No_Cajas := 48, [71].Consec := 193, [71].Envase := 17250, [71].Envases_x_Caja := 1, [71].Densidad_Medida := 0.9148, [71].Linea := 5, [72].Fecha.year := 2021,
        [72].Fecha.Mes := 5, [72].Fecha.Dia := 27, [72].Fecha.Hora := 20, [72].Fecha.Minuto := 42, [72].Fecha.Segundo := 50, [72].Fecha.Milisegundos := 610683, [72].Lote := 147, [72].Operador := 6, [72].Descripcion := 'Aceite Vegetal Torino  Exp.', [72].EAN14 := '17702161820113', [72].QAD := '607020', [72].Peso_Real := 787.0, [72].Peso_Teorico := 786.0, [72].No_Cajas := 48, [72].Consec := 194, [72].Envase := 17250, [72].Envases_x_Caja := 1, [72].Densidad_Medida := 0.9148, [72].Linea := 5, [73].Fecha.year := 2021, [73].Fecha.Mes := 5, [73].Fecha.Dia := 27, [73].Fecha.Hora := 20, [73].Fecha.Minuto := 48, [73].Fecha.Segundo := 14, [73].Fecha.Milisegundos := 628015, [73].Lote := 147, [73].Operador := 6, [73].Descripcion := 'Aceite Vegetal Torino  Exp.', [73].EAN14 := '17702161820113', [73].QAD := '607020', [73].Peso_Real := 789.0, [73].Peso_Teorico := 786.0, [73].No_Cajas := 48, [73].Consec := 195, [73].Envase := 17250, [73].Envases_x_Caja := 1, [73].Densidad_Medida := 0.9148, [73].Linea := 5, [74].Fecha.year := 2021, [74].Fecha.Mes := 5, [74].Fecha.Dia := 27, [74].Fecha.Hora := 20, [74].Fecha.Minuto := 54, [74].Fecha.Segundo := 58, [74].Fecha.Milisegundos := 414231, [74].Lote := 147, [74].Operador := 6, [74].Descripcion := 'Aceite Vegetal Torino  Exp.', [74].EAN14 := '17702161820113', [74].QAD := '607020', [74].Peso_Real := 788.0, [74].Peso_Teorico := 786.0, [74].No_Cajas := 48, [74].Consec := 196, [74].Envase := 17250, [74].Envases_x_Caja := 1, [74].Densidad_Medida := 0.9148, [74].Linea := 5, [75].Fecha.year := 2021,
        [75].Fecha.Mes := 5, [75].Fecha.Dia := 27, [75].Fecha.Hora := 21, [75].Fecha.Minuto := 1, [75].Fecha.Segundo := 21, [75].Fecha.Milisegundos := 319569, [75].Lote := 147, [75].Operador := 6, [75].Descripcion := 'Aceite Vegetal Torino  Exp.', [75].EAN14 := '17702161820113', [75].QAD := '607020', [75].Peso_Real := 787.0, [75].Peso_Teorico := 786.0, [75].No_Cajas := 48, [75].Consec := 197, [75].Envase := 17250, [75].Envases_x_Caja := 1, [75].Densidad_Medida := 0.9148, [75].Linea := 5, [76].Fecha.year := 2021, [76].Fecha.Mes := 5, [76].Fecha.Dia := 27, [76].Fecha.Hora := 21, [76].Fecha.Minuto := 7, [76].Fecha.Segundo := 25, [76].Fecha.Milisegundos := 131378, [76].Lote := 147, [76].Operador := 6, [76].Descripcion := 'Aceite Vegetal Torino  Exp.', [76].EAN14 := '17702161820113', [76].QAD := '607020', [76].Peso_Real := 786.0, [76].Peso_Teorico := 786.0, [76].No_Cajas := 48, [76].Consec := 198, [76].Envase := 17250, [76].Envases_x_Caja := 1, [76].Densidad_Medida := 0.9148, [76].Linea := 5, [77].Fecha.year := 2021, [77].Fecha.Mes := 5, [77].Fecha.Dia := 27, [77].Fecha.Hora := 21, [77].Fecha.Minuto := 12, [77].Fecha.Segundo := 42, [77].Fecha.Milisegundos := 644403, [77].Lote := 147, [77].Operador := 6, [77].Descripcion := 'Aceite Vegetal Torino  Exp.', [77].EAN14 := '17702161820113', [77].QAD := '607020', [77].Peso_Real := 787.0, [77].Peso_Teorico := 786.0, [77].No_Cajas := 48, [77].Consec := 199, [77].Envase := 17250, [77].Envases_x_Caja := 1, [77].Densidad_Medida := 0.9148, [77].Linea := 5, [78].Fecha.year := 2021,
        [78].Fecha.Mes := 5, [78].Fecha.Dia := 27, [78].Fecha.Hora := 21, [78].Fecha.Minuto := 18, [78].Fecha.Segundo := 26, [78].Fecha.Milisegundos := 502578, [78].Lote := 147, [78].Operador := 6, [78].Descripcion := 'Aceite Vegetal Torino  Exp.', [78].EAN14 := '17702161820113', [78].QAD := '607020', [78].Peso_Real := 788.0, [78].Peso_Teorico := 786.0, [78].No_Cajas := 48, [78].Consec := 200, [78].Envase := 17250, [78].Envases_x_Caja := 1, [78].Densidad_Medida := 0.9148, [78].Linea := 5, [79].Fecha.year := 2021, [79].Fecha.Mes := 5, [79].Fecha.Dia := 27, [79].Fecha.Hora := 21, [79].Fecha.Minuto := 25, [79].Fecha.Segundo := 29, [79].Fecha.Milisegundos := 869378, [79].Lote := 147, [79].Operador := 6, [79].Descripcion := 'Aceite Vegetal Torino  Exp.', [79].EAN14 := '17702161820113', [79].QAD := '607020', [79].Peso_Real := 787.0, [79].Peso_Teorico := 786.0, [79].No_Cajas := 48, [79].Consec := 201, [79].Envase := 17250, [79].Envases_x_Caja := 1, [79].Densidad_Medida := 0.9148, [79].Linea := 5, [80].Fecha.year := 2021, [80].Fecha.Mes := 5, [80].Fecha.Dia := 27, [80].Fecha.Hora := 21, [80].Fecha.Minuto := 30, [80].Fecha.Segundo := 9, [80].Fecha.Milisegundos := 920967, [80].Lote := 147, [80].Operador := 6, [80].Descripcion := 'Aceite Vegetal Torino  Exp.', [80].EAN14 := '17702161820113', [80].QAD := '607020', [80].Peso_Real := 787.0, [80].Peso_Teorico := 786.0, [80].No_Cajas := 48, [80].Consec := 202, [80].Envase := 17250, [80].Envases_x_Caja := 1, [80].Densidad_Medida := 0.9148, [80].Linea := 5, [81].Fecha.year := 2021,
        [81].Fecha.Mes := 5, [81].Fecha.Dia := 27, [81].Fecha.Hora := 21, [81].Fecha.Minuto := 37, [81].Fecha.Segundo := 33, [81].Fecha.Milisegundos := 559268, [81].Lote := 147, [81].Operador := 6, [81].Descripcion := 'Aceite Vegetal Torino  Exp.', [81].EAN14 := '17702161820113', [81].QAD := '607020', [81].Peso_Real := 787.0, [81].Peso_Teorico := 786.0, [81].No_Cajas := 48, [81].Consec := 203, [81].Envase := 17250, [81].Envases_x_Caja := 1, [81].Densidad_Medida := 0.9148, [81].Linea := 5, [82].Fecha.year := 2021, [82].Fecha.Mes := 5, [82].Fecha.Dia := 27, [82].Fecha.Hora := 21, [82].Fecha.Minuto := 43, [82].Fecha.Segundo := 55, [82].Fecha.Milisegundos := 778548, [82].Lote := 147, [82].Operador := 6, [82].Descripcion := 'Aceite Vegetal Torino  Exp.', [82].EAN14 := '17702161820113', [82].QAD := '607020', [82].Peso_Real := 789.0, [82].Peso_Teorico := 786.0, [82].No_Cajas := 48, [82].Consec := 204, [82].Envase := 17250, [82].Envases_x_Caja := 1, [82].Densidad_Medida := 0.9148, [82].Linea := 5, [83].Fecha.year := 2021, [83].Fecha.Mes := 5, [83].Fecha.Dia := 27, [83].Fecha.Hora := 21, [83].Fecha.Minuto := 49, [83].Fecha.Segundo := 50, [83].Fecha.Milisegundos := 468922, [83].Lote := 147, [83].Operador := 6, [83].Descripcion := 'Aceite Vegetal Torino  Exp.', [83].EAN14 := '17702161820113', [83].QAD := '607020', [83].Peso_Real := 789.0, [83].Peso_Teorico := 786.0, [83].No_Cajas := 48, [83].Consec := 205, [83].Envase := 17250, [83].Envases_x_Caja := 1, [83].Densidad_Medida := 0.9148, [83].Linea := 5, [84].Fecha.year := 2021,
        [84].Fecha.Mes := 5, [84].Fecha.Dia := 27, [84].Fecha.Hora := 21, [84].Fecha.Minuto := 55, [84].Fecha.Segundo := 48, [84].Fecha.Milisegundos := 524597, [84].Lote := 147, [84].Operador := 6, [84].Descripcion := 'Aceite Vegetal Torino  Exp.', [84].EAN14 := '17702161820113', [84].QAD := '607020', [84].Peso_Real := 788.0, [84].Peso_Teorico := 786.0, [84].No_Cajas := 48, [84].Consec := 206, [84].Envase := 17250, [84].Envases_x_Caja := 1, [84].Densidad_Medida := 0.9148, [84].Linea := 5, [85].Fecha.year := 2021, [85].Fecha.Mes := 5, [85].Fecha.Dia := 27, [85].Fecha.Hora := 22, [85].Fecha.Minuto := 1, [85].Fecha.Segundo := 56, [85].Fecha.Milisegundos := 647666, [85].Lote := 147, [85].Operador := 6, [85].Descripcion := 'Aceite Vegetal Torino  Exp.', [85].EAN14 := '17702161820113', [85].QAD := '607020', [85].Peso_Real := 788.0, [85].Peso_Teorico := 786.0, [85].No_Cajas := 48, [85].Consec := 207, [85].Envase := 17250, [85].Envases_x_Caja := 1, [85].Densidad_Medida := 0.9148, [85].Linea := 5, [86].Fecha.year := 2021, [86].Fecha.Mes := 5, [86].Fecha.Dia := 27, [86].Fecha.Hora := 22, [86].Fecha.Minuto := 7, [86].Fecha.Segundo := 15, [86].Fecha.Milisegundos := 55253, [86].Lote := 147, [86].Operador := 6, [86].Descripcion := 'Aceite Vegetal Torino  Exp.', [86].EAN14 := '17702161820113', [86].QAD := '607020', [86].Peso_Real := 793.0, [86].Peso_Teorico := 786.0, [86].No_Cajas := 48, [86].Consec := 208, [86].Envase := 17250, [86].Envases_x_Caja := 1, [86].Densidad_Medida := 0.9148, [86].Linea := 5, [87].Fecha.year := 2021,
        [87].Fecha.Mes := 5, [87].Fecha.Dia := 27, [87].Fecha.Hora := 22, [87].Fecha.Minuto := 12, [87].Fecha.Segundo := 57, [87].Fecha.Milisegundos := 864929, [87].Lote := 147, [87].Operador := 6, [87].Descripcion := 'Aceite Vegetal Torino  Exp.', [87].EAN14 := '17702161820113', [87].QAD := '607020', [87].Peso_Real := 787.0, [87].Peso_Teorico := 786.0, [87].No_Cajas := 48, [87].Consec := 209, [87].Envase := 17250, [87].Envases_x_Caja := 1, [87].Densidad_Medida := 0.9148, [87].Linea := 5, [88].Fecha.year := 2021, [88].Fecha.Mes := 5, [88].Fecha.Dia := 27, [88].Fecha.Hora := 22, [88].Fecha.Minuto := 17, [88].Fecha.Segundo := 47, [88].Fecha.Milisegundos := 795924, [88].Lote := 147, [88].Operador := 6, [88].Descripcion := 'Aceite Vegetal Torino  Exp.', [88].EAN14 := '17702161820113', [88].QAD := '607020', [88].Peso_Real := 788.0, [88].Peso_Teorico := 786.0, [88].No_Cajas := 48, [88].Consec := 210, [88].Envase := 17250, [88].Envases_x_Caja := 1, [88].Densidad_Medida := 0.9148, [88].Linea := 5, [89].Fecha.year := 2021, [89].Fecha.Mes := 5, [89].Fecha.Dia := 27, [89].Fecha.Hora := 22, [89].Fecha.Minuto := 22, [89].Fecha.Segundo := 51, [89].Fecha.Milisegundos := 894640, [89].Lote := 147, [89].Operador := 6, [89].Descripcion := 'Aceite Vegetal Torino  Exp.', [89].EAN14 := '17702161820113', [89].QAD := '607020', [89].Peso_Real := 788.0, [89].Peso_Teorico := 786.0, [89].No_Cajas := 48, [89].Consec := 211, [89].Envase := 17250, [89].Envases_x_Caja := 1, [89].Densidad_Medida := 0.9148, [89].Linea := 5, [90].Fecha.year := 2021,
        [90].Fecha.Mes := 5, [90].Fecha.Dia := 27, [90].Fecha.Hora := 22, [90].Fecha.Minuto := 27, [90].Fecha.Segundo := 44, [90].Fecha.Milisegundos := 226445, [90].Lote := 147, [90].Operador := 6, [90].Descripcion := 'Aceite Vegetal Torino  Exp.', [90].EAN14 := '17702161820113', [90].QAD := '607020', [90].Peso_Real := 787.0, [90].Peso_Teorico := 786.0, [90].No_Cajas := 48, [90].Consec := 212, [90].Envase := 17250, [90].Envases_x_Caja := 1, [90].Densidad_Medida := 0.9148, [90].Linea := 5, [91].Fecha.year := 2021, [91].Fecha.Mes := 5, [91].Fecha.Dia := 27, [91].Fecha.Hora := 22, [91].Fecha.Minuto := 35, [91].Fecha.Segundo := 5, [91].Fecha.Milisegundos := 374951, [91].Lote := 147, [91].Operador := 6, [91].Descripcion := 'Aceite Vegetal Torino  Exp.', [91].EAN14 := '17702161820113', [91].QAD := '607020', [91].Peso_Real := 788.0, [91].Peso_Teorico := 786.0, [91].No_Cajas := 48, [91].Consec := 213, [91].Envase := 17250, [91].Envases_x_Caja := 1, [91].Densidad_Medida := 0.9148, [91].Linea := 5, [92].Fecha.year := 2021, [92].Fecha.Mes := 5, [92].Fecha.Dia := 27, [92].Fecha.Hora := 22, [92].Fecha.Minuto := 42, [92].Fecha.Segundo := 12, [92].Fecha.Milisegundos := 904782, [92].Lote := 147, [92].Operador := 6, [92].Descripcion := 'Aceite Vegetal Torino  Exp.', [92].EAN14 := '17702161820113', [92].QAD := '607020', [92].Peso_Real := 789.0, [92].Peso_Teorico := 786.0, [92].No_Cajas := 48, [92].Consec := 214, [92].Envase := 17250, [92].Envases_x_Caja := 1, [92].Densidad_Medida := 0.9148, [92].Linea := 5, [93].Fecha.year := 2021,
        [93].Fecha.Mes := 5, [93].Fecha.Dia := 27, [93].Fecha.Hora := 22, [93].Fecha.Minuto := 47, [93].Fecha.Segundo := 23, [93].Fecha.Milisegundos := 229821, [93].Lote := 147, [93].Operador := 6, [93].Descripcion := 'Aceite Vegetal Torino  Exp.', [93].EAN14 := '17702161820113', [93].QAD := '607020', [93].Peso_Real := 788.0, [93].Peso_Teorico := 786.0, [93].No_Cajas := 48, [93].Consec := 215, [93].Envase := 17250, [93].Envases_x_Caja := 1, [93].Densidad_Medida := 0.9148, [93].Linea := 5, [94].Fecha.year := 2021, [94].Fecha.Mes := 5, [94].Fecha.Dia := 27, [94].Fecha.Hora := 22, [94].Fecha.Minuto := 52, [94].Fecha.Segundo := 46, [94].Fecha.Milisegundos := 173212, [94].Lote := 147, [94].Operador := 6, [94].Descripcion := 'Aceite Vegetal Torino  Exp.', [94].EAN14 := '17702161820113', [94].QAD := '607020', [94].Peso_Real := 787.0, [94].Peso_Teorico := 786.0, [94].No_Cajas := 48, [94].Consec := 216, [94].Envase := 17250, [94].Envases_x_Caja := 1, [94].Densidad_Medida := 0.9148, [94].Linea := 5, [95].Fecha.year := 2021, [95].Fecha.Mes := 5, [95].Fecha.Dia := 27, [95].Fecha.Hora := 23, [95].Fecha.Minuto := 3, [95].Fecha.Segundo := 8, [95].Fecha.Milisegundos := 268358, [95].Lote := 147, [95].Operador := 6, [95].Descripcion := 'Aceite Vegetal Torino  Exp.', [95].EAN14 := '17702161820113', [95].QAD := '607020', [95].Peso_Real := 706.0, [95].Peso_Teorico := 704.0, [95].No_Cajas := 43, [95].Consec := 217, [95].Envase := 17250, [95].Envases_x_Caja := 1, [95].Densidad_Medida := 0.9148, [95].Linea := 5);
   Cola_Impresion_Vacia : UDT_COLA;
   Cola_Peso_Bidones : REAL[50];
   Cola_Peso_Caja_Bidon_Ayer : REAL[50];
   Cola_Peso_Caja_Elmar : REAL[50];
   Cola_Peso_Caja_Elmar_Ayer : REAL[50];
   Cola_Peso_Caja_Fogg1 : REAL[50];
   Cola_Peso_Caja_Fogg1_Ayer : REAL[50];
   Cola_Peso_Caja_Fogg2 : REAL[50];
   Cola_Peso_Caja_Fogg2_Ayer : REAL[50];
   Cola_Peso_Caja_Karat : REAL[50];
   Cola_Peso_Caja_Karat_Ayer : REAL[50];
   Cola_QAD_Densidad_Bidon_Ayer : STRING[50];
   Cola_QAD_Densidad_Bidones : STRING[50];
   Cola_QAD_Densidad_Elmar : STRING[50];
   Cola_QAD_Densidad_Elmar_Ayer : STRING[50];
   Cola_QAD_Densidad_Fogg1 : STRING[50];
   Cola_QAD_Densidad_Fogg1_Ayer : STRING[50];
   Cola_QAD_Densidad_Fogg2 : STRING[50];
   Cola_QAD_Densidad_Fogg2_Ayer : STRING[50];
   Cola_QAD_Densidad_Karat : STRING[50];
   Cola_QAD_Densidad_Karat_Ayer : STRING[50];
   Consecutivo : INT := 110;
   Consecutivo_2 : INT := 17;
   Consecutivo_String : Consecutivo := (Consec[0] := '110', Consec[1] := '99', Consec[2] := '9');
   Consolidado_Est : UDT_COLA[50] := ([20].Lote := 46, [20].Descripcion := 'Sarita  vegetal Caja 24 x 400 cm3', [20].QAD := '627500', [20].Peso_Real := 28001.0, [20].Peso_Teorico := 28197.0, [20].No_Cajas := 2969, [21].Lote := 21, [21].Descripcion := 'Sarita  vegetal Caja 12 x 750 cm3', [21].QAD := '627300', [21].Peso_Real := 12603.0, [21].Peso_Teorico := 12728.0, [21].No_Cajas := 1444);
   Cont_Prod_1 : DINT := 23;
   Cont_Prod_2 : DINT := 112;
   Cont_Prod_3 : DINT := 23;
   Cont_Prod_4 : DINT := 117;
   Contador_Consecutivo : COUNTER := (PRE := 5000, ACC := 110);
   Control_Cola_Est1 : CONTROL := (LEN := 100, EM := 1);
   Control_Cola_Est2 : CONTROL := (LEN := 100, POS := 57);
   Control_Cola_Est3 : CONTROL := (LEN := 100, EM := 1);
   Control_Cola_Est4 : CONTROL := (LEN := 100, POS := 53);
   Control_Densidad_Bidones : CONTROL := (LEN := 50, EM := 1);
   Control_Densidad_Elmar : CONTROL := (LEN := 50, EM := 1);
   Control_Densidad_Elmar1 : CONTROL := (LEN := 5, EM := 1);
   Control_Densidad_Fogg1 : CONTROL := (LEN := 50, EM := 1);
   Control_Densidad_Fogg2 : CONTROL := (LEN := 50, EM := 1);
   Control_Densidad_Karat : CONTROL := (LEN := 50, EM := 1);
   Control_Peso_Caja_Elmar : CONTROL := (LEN := 10, EM := 1);
   Control_Salida_Est1 : CONTROL;
   Counter_R_Estacion1 : COUNTER := (PRE := 50);
   Counter_R_Estacion2 : COUNTER := (PRE := 50);
   Counter_R_Estacion3 : COUNTER := (PRE := 20, ACC := 1);
   Counter_R_Estacion4 : COUNTER := (PRE := 20);
   CUATRO : SINT := 4;
   Datos_1_Manual : BOOL;
   Datos_2_Manual : BOOL;
   Datos_3_Manual : BOOL;
   Datos_4_Manual : BOOL;
   Datos_Leidos_Scanner : QR := (LEN := 112);
   Densidad_1 : REAL := 0.9152;
   Densidad_2 : REAL := 0.9152;
   Densidad_3 : REAL := 0.9152;
   Densidad_4 : REAL := 0.9148;
   Densidad_Bidon : REAL;
   Densidad_Bidon_1 : REAL := 0.9148;
   Densidad_Bidones : REAL;
   Densidad_Bidones_1 : REAL;
   Densidad_Bidones_OK : BOOL;
   Densidad_Elmar : REAL;
   Densidad_Elmar_1 : REAL := 0.9152;
   Densidad_Elmar_OK : BOOL;
   Densidad_Fogg1 : REAL;
   Densidad_Fogg1_1 : REAL := 0.9139;
   Densidad_Fogg1_OK : BOOL;
   Densidad_Fogg2 : REAL;
   Densidad_Fogg2_1 : REAL := 0.9152;
   Densidad_Fogg2_OK : BOOL;
   Densidad_Karat : REAL;
   Densidad_Karat_1 : REAL;
   Densidad_Karat_OK : BOOL;
   Dia_del_Ano : INT := 148;
   Dia_Year : DINT;
   Diff_Peso_1 : DINT := 858;
   Diff_Peso_2 : DINT := 578;
   Diff_Peso_3 : DINT := 857;
   Diff_Peso_4 : DINT := 746;
   DM8000_DMCC_Command : STRING;   // A DMCC Command to send to the DM8000
   DM8000_DMCC_Enable : BOOL;
   DM8000_Read_Enable : BOOL := 1;
   DM8000_Read_Results : STRING;   // A string containing the results of a data read from the DM8000
   DOS : SINT := 2;
   EAN14_1 : Codigo_Barras := '17702161567070';
   EAN14_2 : Codigo_Barras := '17702161409646';
   EAN14_3 : Codigo_Barras := '17702161567070';
   EAN14_4 : Codigo_Barras := '17702161820113';
   ENTRE_No_CAJAS_1 : DINT;
   ENTRE_No_CAJAS_2 : DINT;
   ENTRE_No_CAJAS_3 : DINT;
   Espacios : STRING := '                                                  ';
   ESTACION_1 : DINT := 1;
   Estacion_1_Cajas : UDT_CAJAS := (No_Cajas[0] := '36', No_Cajas[1] := '2');
   Estacion_1_EAN14 : UDT_EAN14 := (EAN14 := '67702179402405');
   Estacion_1_GCola : UDT_COLA := (Fecha.year := 2020, Fecha.Mes := 11, Fecha.Dia := 7, Fecha.Hora := 12, Fecha.Minuto := 2, Fecha.Segundo := 46, Fecha.Milisegundos := 11719, Lote := 312, Operador := 5, Descripcion := 'Oriental 100% ole$EDna x 3000 ML  Cj 6 Und', EAN14 := '17702161567070', QAD := '605990', Peso_Real := 858.0, Peso_Teorico := 865.0, No_Cajas := 50, Consec := 22, Envase := 3000, Envases_x_Caja := 6, Densidad_Medida := 0.9152, Linea := 3);
   Estacion_1_GCola_1 : UDT_COLA := (Fecha.year := 2021, Fecha.Mes := 5, Fecha.Dia := 28, Fecha.Hora := 16, Fecha.Minuto := 19, Fecha.Segundo := 37, Fecha.Milisegundos := 137377, Lote := 148, Operador := 5, Descripcion := 'Oriental 100% ole$EDna x 3000 ML  Cj 6 Und', EAN14 := '17702161567070', QAD := '605990', Peso_Real := -23.0, Peso_Teorico := 865.0, No_Cajas := 50, Consec := 22, Envase := 3000, Envases_x_Caja := 6, Densidad_Medida := 0.9152, Linea := 3);
   Estacion_1_General : UDT_GENERAL := (dd[0] := '28', dd[1] := '9', mm[0] := '0', mm[1] := '5', yy[0] := '2021', hh[0] := '16', hh[1] := '9', min[0] := '19', min[1] := '9', lote[0] := '0', lote[1] := '99', lote[2] := '148', clima := '0', operador[0] := '0', operador[1] := '5', Descripcion := 'Oriental 100% ole$EDna x 3000 ML  Cj 6 Und', QAD := '605990', Peso_Real[0] := '0', Peso_Real[1] := '0', Peso_Real[2] := '-23', Peso_Teorico[0] := '865', Peso_Teorico[1] := '12', Peso_Teorico[2] := '0', No_Cajas[0] := '0', No_Cajas[1] := '50', No_Cajas[2] := '0');
   Estacion_1_Inicia_Conteo : BOOL := 1;
   Estacion_1_PReal : UDT_PESO_REAL := (Peso_Real[0] := '0', Peso_Real[1] := '-23');
   Estacion_1_PTeorico : UDT_PESO_TEORICO := (Peso_Teorico[0] := '698', Peso_Teorico[1] := '39');
   Estacion_1_QAD : UDT_QAD := (Codigo := '40240');
   Estacion_1_Resumen : UDT_COLA[20] := ([0].Descripcion := 'Oriental 100% ole$EDna x 3000 ML  Cj 6 Und', [0].QAD := '605990');
   Estacion_1_Resumen_A : UDT_COLA[20] := ([0].Descripcion := 'Oriental 100% ole$EDna x 3000 ML  Cj 6 Und', [0].QAD := '605990');
   Estacion_1_String : STRING := '1';
   ESTACION_2 : DINT := 2;
   Estacion_2_GCola : UDT_COLA := (Fecha.year := 2021, Fecha.Mes := 5, Fecha.Dia := 28, Fecha.Hora := 14, Fecha.Minuto := 42, Fecha.Segundo := 25, Fecha.Milisegundos := 529661, Lote := 148, Operador := 5, Descripcion := 'Alegria Caja 12 x 900 cm3  - Costa', EAN14 := '17702161409646', QAD := '600620', Peso_Real := 548.0, Peso_Teorico := 543.0, No_Cajas := 52, Consec := 109, Envase := 900, Envases_x_Caja := 12, Densidad_Medida := 0.9152, Linea := 1);
   Estacion_2_GCola_1 : UDT_COLA := (Fecha.year := 2021, Fecha.Mes := 5, Fecha.Dia := 28, Fecha.Hora := 16, Fecha.Minuto := 19, Fecha.Segundo := 41, Fecha.Milisegundos := 243088, Lote := 148, Operador := 5, Descripcion := 'Alegria Caja 12 x 900 cm3  - Costa', EAN14 := '17702161409646', QAD := '600620', Peso_Real := -30.0, Peso_Teorico := 585.0, No_Cajas := 56, Consec := 109, Envase := 900, Envases_x_Caja := 12, Densidad_Medida := 0.9152, Linea := 1);
   Estacion_2_General : UDT_GENERAL := (dd[0] := '0', dd[1] := '9', mm[0] := '10', mm[1] := '9', yy[0] := '2017', hh[0] := '16', hh[1] := '9', min[0] := '0', min[1] := '9', lote[0] := '282', clima := '0', operador[0] := '0', operador[1] := '5', Descripcion := 'Alegria Caja 12 x 900 cm3  - Costa', QAD := '600620', Peso_Real[0] := '0', Peso_Real[1] := '0', Peso_Real[2] := '-30', Peso_Teorico[0] := '585', Peso_Teorico[1] := '31', Peso_Teorico[2] := '0', No_Cajas[0] := '0', No_Cajas[1] := '56', No_Cajas[2] := '3');
   Estacion_2_PRT : UDT_GENERAL := (dd[0] := '13', mm[0] := '0', mm[1] := '9', yy[0] := '2017', hh[0] := '17', hh[1] := '11', min[0] := '0', min[1] := '0', lote[0] := '255', clima := '0', operador[0] := '0', operador[1] := '5', Descripcion := 'Esta es la descripcion de nuestro de los aceite   ');
   Estacion_2_Resumen : UDT_COLA[20] := ([0].Lote := 57, [0].Descripcion := 'Alegria Caja 12 x 900 cm3  - Costa', [0].QAD := '600620', [0].Peso_Real := 33573.0, [0].Peso_Teorico := 33303.0, [0].No_Cajas := 3188);
   Estacion_2_Resumen_A : UDT_COLA[20] := ([0].Descripcion := 'Mazorca de Oro Caja 12 x 1000 cm3', [0].QAD := '605150', [1].Lote := 62, [1].Descripcion := 'Alegria Caja 12 x 900 cm3  - Costa', [1].QAD := '600620', [1].Peso_Real := 35437.0, [1].Peso_Teorico := 35288.0, [1].No_Cajas := 3378);
   Estacion_2_String : STRING := '2';
   ESTACION_3 : DINT := 3;
   Estacion_3_GCola : UDT_COLA := (Fecha.year := 2021, Fecha.Mes := 5, Fecha.Dia := 27, Fecha.Hora := 20, Fecha.Minuto := 7, Fecha.Segundo := 7, Fecha.Milisegundos := 884753, Lote := 147, Operador := 5, Descripcion := 'Alegria Caja 6 x 3000 cm3  - Costa', EAN14 := '17702161043987', QAD := '600300', Peso_Real := 52.0, Peso_Teorico := 52.0, No_Cajas := 3, Consec := 192, Envase := 3000, Envases_x_Caja := 6, Densidad_Medida := 0.9152, Linea := 3);
   Estacion_3_GCola_1 : UDT_COLA := (Fecha.year := 2021, Fecha.Mes := 5, Fecha.Dia := 28, Fecha.Hora := 16, Fecha.Minuto := 19, Fecha.Segundo := 39, Fecha.Milisegundos := 793548, Lote := 148, Operador := 5, Descripcion := 'Oriental 100% oleina x 3000 ML  Cj 6 Und', EAN14 := '17702161567070', QAD := '605990', Peso_Teorico := 865.0, No_Cajas := 50, Consec := 192, Envase := 3000, Envases_x_Caja := 6, Densidad_Medida := 0.9152, Linea := 3);
   Estacion_3_General : UDT_GENERAL := (dd[0] := '0', dd[1] := '9', mm[0] := '10', mm[1] := '9', yy[0] := '2017', hh[0] := '16', hh[1] := '9', min[0] := '0', min[1] := '9', lote[0] := '282', clima := '0', operador[0] := '0', operador[1] := '5', Descripcion := 'Oriental 100% oleina x 3000 ML  Cj 6 Und', QAD := '605990', Peso_Real[0] := '0', Peso_Real[1] := '0', Peso_Real[2] := '0', Peso_Teorico[0] := '865', Peso_Teorico[1] := '52', Peso_Teorico[2] := '0', No_Cajas[0] := '0', No_Cajas[1] := '50', No_Cajas[2] := '3');
   Estacion_3_PRT : UDT_GENERAL := (dd[0] := '13', mm[0] := '0', mm[1] := '9', yy[0] := '2017', hh[0] := '17', hh[1] := '11', min[0] := '0', min[1] := '0', lote[0] := '255', clima := '0', operador[0] := '0', operador[1] := '5', Descripcion := 'Esta es la descripcion de nuestro de los aceite   ');
   Estacion_3_Resumen : UDT_COLA[20] := ([0].Descripcion := 'Alegria Caja 6 x 3000 cm3  - Costa', [0].QAD := '600300', [1].Descripcion := 'Oriental 100% oleina x 3000 ML  Cj 6 Und', [1].QAD := '605990');
   Estacion_3_Resumen_A : UDT_COLA[20] := ([0].Descripcion := 'Mazorca de Oro Caja 6 x 3000 cm3', [0].QAD := '604850', [1].Descripcion := 'Alegria Caja 6 x 3000 cm3  - Costa', [1].QAD := '600300', [2].Lote := 1, [2].Descripcion := 'La Muneca Comisariato Caja 6 x 3000 cm3', [2].QAD := '602800', [2].Peso_Real := 207.0, [2].Peso_Teorico := 207.0, [2].No_Cajas := 12, [3].Lote := 58, [3].Descripcion := 'Alegria Caja 6 x 3000 cm3  - Costa', [3].QAD := '600300', [3].Peso_Real := 29530.0, [3].Peso_Teorico := 29635.0, [3].No_Cajas := 1713);
   Estacion_3_String : STRING := '3';
   ESTACION_4 : DINT := 4;
   Estacion_4_Cajas : UDT_CAJAS := (No_Cajas[0] := '36', No_Cajas[1] := '2');
   Estacion_4_GCola : UDT_COLA := (Fecha.year := 2021, Fecha.Mes := 5, Fecha.Dia := 28, Fecha.Hora := 14, Fecha.Minuto := 49, Fecha.Segundo := 25, Fecha.Milisegundos := 216916, Lote := 148, Operador := 6, Descripcion := 'Aceite Vegetal Torino  Exp.', EAN14 := '17702161820113', QAD := '607020', Peso_Real := 787.0, Peso_Teorico := 786.0, No_Cajas := 48, Consec := 110, Envase := 17250, Envases_x_Caja := 1, Densidad_Medida := 0.9148, Linea := 5);
   Estacion_4_GCola_1 : UDT_COLA := (Fecha.year := 2021, Fecha.Mes := 5, Fecha.Dia := 28, Fecha.Hora := 16, Fecha.Minuto := 19, Fecha.Segundo := 39, Fecha.Milisegundos := 738083, Lote := 148, Operador := 6, Descripcion := 'Aceite Vegetal Torino  Exp.', EAN14 := '17702161820113', QAD := '607020', Peso_Real := -23.0, Peso_Teorico := 786.0, No_Cajas := 48, Consec := 110, Envase := 17250, Envases_x_Caja := 1, Densidad_Medida := 0.9148, Linea := 5);
   Estacion_4_General : UDT_GENERAL := (clima := '0', operador[0] := '0', operador[1] := '6', Descripcion := 'Aceite Vegetal Torino  Exp.', QAD := '607020', Peso_Real[0] := '0', Peso_Real[1] := '0', Peso_Real[2] := '-23', Peso_Teorico[0] := '786', Peso_Teorico[1] := '33', No_Cajas[0] := '0', No_Cajas[1] := '48', No_Cajas[2] := '2');
   Estacion_4_Resumen : UDT_COLA[20] := ([0].Lote := 53, [0].Descripcion := 'Aceite Vegetal Torino  Exp.', [0].QAD := '607020', [0].Peso_Real := 41779.0, [0].Peso_Teorico := 41658.0, [0].No_Cajas := 2544);
   Estacion_4_Resumen_A : UDT_COLA[20] := ([0].Lote := 96, [0].Descripcion := 'Aceite Vegetal Torino  Exp.', [0].QAD := '607020', [0].Peso_Real := 75610.0, [0].Peso_Teorico := 75374.0, [0].No_Cajas := 4603);
   Estacion_4_String : STRING := '4';
   Ethernet_Duplex_OK : BOOL := 1;
   Ethernet_Duplex_State : ALIAS FOR Ethernet_Module_Status.1;
   Ethernet_Hardware_Mal : BOOL;
   Ethernet_Hardware_Status : ALIAS FOR Ethernet_Module_Status.6;
   Ethernet_Link_State : ALIAS FOR Ethernet_Module_Status.0;
   Ethernet_Module_Status : DINT := 47;
   ETHERNET_STATUS : Ethernet_Status := (EntryStatus[0] := 16384, EntryStatus[1] := 16384, EntryStatus[2] := 16384, EntryStatus[3] := 16384, EntryStatus[4] := 16384, EntryStatus[5] := 16384, EntryStatus[6] := 16384, EntryStatus[7] := 16384, EntryStatus[8] := 16384, EntryStatus[9] := 16384, EntryStatus[10] := 16384, EntryStatus[11] := 16384, EntryStatus[12] := 16384, EntryStatus[13] := 16384, EntryStatus[14] := 16384, EntryStatus[15] := 16384, EntryStatus[16] := 16384, EntryStatus[17] := 16384, EntryStatus[18] := 16384, EntryStatus[19] := 16384, EntryStatus[20] := 16384, EntryStatus[21] := 16384, EntryStatus[22] := 16384, EntryStatus[23] := 16384, EntryStatus[24] := 16384, EntryStatus[25] := 16384, EntryStatus[26] := 16384, EntryStatus[27] := 16384, EntryStatus[28] := 16384, EntryStatus[29] := 16384, EntryStatus[30] := 16384, EntryStatus[31] := 16384, EntryStatus[32] := 16384, EntryStatus[33] := 16384, EntryStatus[34] := 16384, EntryStatus[35] := 16384, EntryStatus[36] := 16384, EntryStatus[37] := 16384, EntryStatus[38] := 16384, EntryStatus[39] := 16384, EntryStatus[40] := 16384, EntryStatus[41] := 16384, EntryStatus[42] := 16384, EntryStatus[43] := 16384, EntryStatus[44] := 16384, EntryStatus[45] := 16384, EntryStatus[46] := 16384, EntryStatus[47] := 16384, EntryStatus[48] := 16384, EntryStatus[49] := 16384, EntryStatus[50] := 16384, EntryStatus[51] := 16384, EntryStatus[52] := 16384, EntryStatus[53] := 16384, EntryStatus[54] := 16384, EntryStatus[55] := 16384, EntryStatus[56] := 16384, EntryStatus[57] := 16384, EntryStatus[58] := 16384, EntryStatus[59] := 16384,
        EntryStatus[60] := 16384, EntryStatus[61] := 16384, EntryStatus[62] := 16384, EntryStatus[63] := 16384, EntryStatus[64] := 16384, EntryStatus[65] := 16384, EntryStatus[66] := 16384, EntryStatus[67] := 16384, EntryStatus[68] := 16384, EntryStatus[69] := 16384, EntryStatus[70] := 16384, EntryStatus[71] := 16384, EntryStatus[72] := 16384, EntryStatus[73] := 16384, EntryStatus[74] := 16384, EntryStatus[75] := 16384, EntryStatus[76] := 16384, EntryStatus[77] := 16384, EntryStatus[78] := 16384, EntryStatus[79] := 16384, EntryStatus[80] := 16384, EntryStatus[81] := 16384, EntryStatus[82] := 16384, EntryStatus[83] := 16384, EntryStatus[84] := 16384, EntryStatus[85] := 16384, EntryStatus[86] := 16384, EntryStatus[87] := 16384, EntryStatus[88] := 16384, EntryStatus[89] := 16384, EntryStatus[90] := 16384, EntryStatus[91] := 16384, EntryStatus[92] := 16384, EntryStatus[93] := 16384, EntryStatus[94] := 16384, EntryStatus[95] := 16384, EntryStatus[96] := 16384, EntryStatus[97] := 16384, EntryStatus[98] := 16384, EntryStatus[99] := 16384, EntryStatus[100] := 16384, EntryStatus[101] := 16384, EntryStatus[102] := 16384, EntryStatus[103] := 16384, EntryStatus[104] := 16384, EntryStatus[105] := 16384, EntryStatus[106] := 16384, EntryStatus[107] := 16384, EntryStatus[108] := 16384, EntryStatus[109] := 16384, EntryStatus[110] := 16384, EntryStatus[111] := 16384, EntryStatus[112] := 16384, EntryStatus[113] := 16384, EntryStatus[114] := 16384, EntryStatus[115] := 16384, EntryStatus[116] := 16384, EntryStatus[117] := 16384, EntryStatus[118] := 16384, EntryStatus[119] := 16384,
        EntryStatus[120] := 16384, EntryStatus[121] := 16384, EntryStatus[122] := 16384, EntryStatus[123] := 16384, EntryStatus[124] := 16384, EntryStatus[125] := 16384, EntryStatus[126] := 16384, EntryStatus[127] := 16384, EntryStatus[128] := 16384, EntryStatus[129] := 16384, EntryStatus[130] := 16384, EntryStatus[131] := 16384, EntryStatus[132] := 16384, EntryStatus[133] := 16384, EntryStatus[134] := 16384, EntryStatus[135] := 16384, EntryStatus[136] := 16384, EntryStatus[137] := 16384, EntryStatus[138] := 16384, EntryStatus[139] := 16384, EntryStatus[140] := 16384, EntryStatus[141] := 16384, EntryStatus[142] := 16384, EntryStatus[143] := 16384, EntryStatus[144] := 16384, EntryStatus[145] := 16384, EntryStatus[146] := 16384, EntryStatus[147] := 16384, EntryStatus[148] := 16384, EntryStatus[149] := 16384, EntryStatus[150] := 16384, EntryStatus[151] := 16384, EntryStatus[152] := 16384, EntryStatus[153] := 16384, EntryStatus[154] := 16384, EntryStatus[155] := 16384, EntryStatus[156] := 16384, EntryStatus[157] := 16384, EntryStatus[158] := 16384, EntryStatus[159] := 16384, EntryStatus[160] := 16384, EntryStatus[161] := 16384, EntryStatus[162] := 16384, EntryStatus[163] := 16384, EntryStatus[164] := 16384, EntryStatus[165] := 16384, EntryStatus[166] := 16384, EntryStatus[167] := 16384, EntryStatus[168] := 16384, EntryStatus[169] := 16384, EntryStatus[170] := 16384, EntryStatus[171] := 16384, EntryStatus[172] := 16384, EntryStatus[173] := 16384, EntryStatus[174] := 16384, EntryStatus[175] := 16384, EntryStatus[176] := 16384, EntryStatus[177] := 16384, EntryStatus[178] := 16384, EntryStatus[179] := 16384,
        EntryStatus[180] := 16384, EntryStatus[181] := 16384, EntryStatus[182] := 16384, EntryStatus[183] := 16384, EntryStatus[184] := 16384, EntryStatus[185] := 16384, EntryStatus[186] := 16384, EntryStatus[187] := 16384, EntryStatus[188] := 16384, EntryStatus[189] := 16384, EntryStatus[190] := 16384, EntryStatus[191] := 16384, EntryStatus[192] := 16384, EntryStatus[193] := 16384, EntryStatus[194] := 16384, EntryStatus[195] := 16384, EntryStatus[196] := 16384, EntryStatus[197] := 16384, EntryStatus[198] := 16384, EntryStatus[199] := 16384, EntryStatus[200] := 16384, EntryStatus[201] := 16384, EntryStatus[202] := 16384, EntryStatus[203] := 16384, EntryStatus[204] := 16384, EntryStatus[205] := 16384, EntryStatus[206] := 16384, EntryStatus[207] := 16384, EntryStatus[208] := 16384, EntryStatus[209] := 16384, EntryStatus[210] := 16384, EntryStatus[211] := 16384, EntryStatus[212] := 16384, EntryStatus[213] := 16384, EntryStatus[214] := 16384, EntryStatus[215] := 16384, EntryStatus[216] := 16384, EntryStatus[217] := 16384, EntryStatus[218] := 16384, EntryStatus[219] := 16384, EntryStatus[220] := 16384, EntryStatus[221] := 16384, EntryStatus[222] := 16384, EntryStatus[223] := 16384, EntryStatus[224] := 16384, EntryStatus[225] := 16384, EntryStatus[226] := 16384, EntryStatus[227] := 16384, EntryStatus[228] := 16384, EntryStatus[229] := 16384, EntryStatus[230] := 16384, EntryStatus[231] := 16384, EntryStatus[232] := 16384, EntryStatus[233] := 16384, EntryStatus[234] := 16384, EntryStatus[235] := 16384, EntryStatus[236] := 16384, EntryStatus[237] := 16384, EntryStatus[238] := 16384, EntryStatus[239] := 16384,
        EntryStatus[240] := 16384, EntryStatus[241] := 16384, EntryStatus[242] := 16384, EntryStatus[243] := 16384, EntryStatus[244] := 16384, EntryStatus[245] := 16384, EntryStatus[246] := 16384, EntryStatus[247] := 16384, EntryStatus[248] := 16384, EntryStatus[249] := 16384, EntryStatus[250] := 16384, EntryStatus[251] := 16384, EntryStatus[252] := 16384, EntryStatus[253] := 16384, EntryStatus[254] := 16384, EntryStatus[255] := 16384);
   FLASH_TIMERS : TIMER[2] := ([0].ACC := 68, [0].EN := 1, [0].DN := 1, [1].ACC := 68, [1].EN := 1, [1].DN := 1);
   FORCE_STATUS : DINT;
   Forx : SINT := 2;
   Fory : SINT := 10;
   Forz : SINT;
   found : SINT;
   Get_Ethernet_Module_Link_Status : MESSAGE;
   Hardy_Basculas_Net_OK : BOOL := 1;
   Hora_Ingreso_Datos_Elmar : Hora_y_Fecha := (year := 2020, Mes := 5, Dia := 21, Hora := 17, Minuto := 3, Segundo := 26, Milisegundos := 553850);
   Hoy : DINT := 148;
   Impreso_1 : BOOL;
   Impreso_2 : BOOL;
